// TwinCAT 3 PLC project PLC
// ProgramVersion: 3.1.4023.0
// libraries:
//   Tc2_Standard, * (Beckhoff Automation GmbH)
//   Tc2_System, * (Beckhoff Automation GmbH)
//   Tc3_Module, * (Beckhoff Automation GmbH)
// project tree:
//   / PlcTask.TcTTO
//   POUs/ MAIN.TcPOU
//   DUTs/IO/PdoEntries/ Status_57491DF1.TcDUT, Status_D4FDECD4.TcDUT, Control_0B2F8B70.TcDUT, Status_A3AA621F.TcDUT, Status_B0753356.TcDUT, Status_F2CE6D91.TcDUT, STATUS_B0753356.TcDUT, Status_8F1D55D8.TcDUT, Status_ACC8459F.TcDUT, Status_3A9E406C.TcDUT, Control_D500AB79.TcDUT, Status_D8D782C3.TcDUT, Control_6EF2C5D0.TcDUT, Status_E3E7FD12.TcDUT, Status_8CBE219F.TcDUT, Status_B6795845.TcDUT, Control_5FD4673D.TcDUT, Status_1E008DB9.TcDUT, Status_3035BE2E.TcDUT, Control_F189B737.TcDUT, Control_C948E0F2.TcDUT, Status_51F572C8.TcDUT
//   DUTs/IO/PDOs/ InfoData_6F19DB2B.TcDUT, Channel_830843C1.TcDUT, WcState_9091E0EB.TcDUT, ID_Inputs_07C9D28F.TcDUT, InfoData_32EB74EA.TcDUT, Latch_8E413295.TcDUT, WcState_B516A264.TcDUT, InfoData_A7436BC6.TcDUT, CNT_Input_Channel_FF10BD3C.TcDUT, DIG_Inputs_CAFF6004.TcDUT, DIG_Inputs_Device_1F4E72EB.TcDUT, CNT_Output_Channel_550BB6DF.TcDUT, DIG_Inputs_Channel_ACAA0425.TcDUT, DIG_Inputs_Channel_CC455148.TcDUT, DIG_Inputs_Channel_38F9DD27.TcDUT, AI_Inputs_Channel_C3DE7A0A.TcDUT, DIG_Inputs_Device_B3EA4204.TcDUT, Channel_42CA91F7.TcDUT, WcState_0B2B16F9.TcDUT, Diag_Channel_830843C1.TcDUT, DIG_Inputs_CC455148.TcDUT, DIG_Diag_Inputs_584303BF.TcDUT, DIG_Inputs_Device_E94E5BF9.TcDUT, DIG_Outputs_28AC1A9E.TcDUT, DIG_Outputs_Device_36A5EF17.TcDUT, DIG_Inputs_2D77DD63.TcDUT, DI_Inputs_Channel_91AC31B7.TcDUT, DO_Outputs_Channel_28AC1A9E.TcDUT, DIG_Diag_Inputs_Channel_584303BF.TcDUT, DIG_Output_Channel_28AC1A9E.TcDUT, DIG_Outputs_Channel_28AC1A9E.TcDUT, DIG_Inputs_Device_27CCC866.TcDUT, AI_Standard_Channel_A8DF64E3.TcDUT, RTD_RTDInputs_Channel_A8DF64E3.TcDUT, AI_Standard_Channel_4A394481.TcDUT, Ch1_Status_75824485.TcDUT, Ch1_Sample_A71DD501.TcDUT, Ch2_Status_75824485.TcDUT, Ch2_Sample_9F6886E6.TcDUT, NextSync1Time_9AFDC275.TcDUT, Sample_Count_EA88CAD9.TcDUT, InfoData_BEF6B88E.TcDUT, DIG_Inputs_697E0EF2.TcDUT, AI_Inputs_Channel_45213104.TcDUT, DEV_Inputs_Device_5F4E175E.TcDUT, DIG_Outputs_DE230DD5.TcDUT, DEV_Outputs_Device_59FFD247.TcDUT, AI_Inputs_Channel_5A86716D.TcDUT, AO_Output_Channel_BA7EBB7C.TcDUT, DI_Inputs_1F3A9325.TcDUT, AI_Inputs_Channel_A8DF64E3.TcDUT, SSI_Inputs_0E3D8E33.TcDUT, ENC_Status_compact_F4F89583.TcDUT, ENC_Control_compact_E6DC9B25.TcDUT, ENC_Status_compact_7D3464F3.TcDUT, ENC_Control_compact_21E2D14D.TcDUT, COM_Inputs_6C2FC202.TcDUT, COM_Outputs_5D00B5E7.TcDUT, COM_TxPDO_Map_Inputs_Channel_C252EAC2.TcDUT, COM_RxPDO_Map_Outputs_Channel_B336F4EE.TcDUT, COM_TxPDO_Map_Inputs_Channel_6C2FC202.TcDUT, COM_RxPDO_Map_Outputs_Channel_5D00B5E7.TcDUT, DIS_Inputs_E0E384E3.TcDUT, DIS_Outputs_6C9BFFEE.TcDUT, DeviceState_Inputs_Device_A1210598.TcDUT, DeviceState_Inputs_C7251DC9.TcDUT, Digital_Inputs_83D7E782.TcDUT, InfoData_90184F0C.TcDUT, Module_1_DeviceState_Inputs_Device_5322301C.TcDUT, Module_2_DeviceState_Inputs_B92A0D6A.TcDUT, Module_11_Digital_Inputs_33FD8372.TcDUT, ENC_Status_compact_4D066E1A.TcDUT, STM_Status_36ED096F.TcDUT, STM_Control_BA4CE352.TcDUT, STM_Velocity_A47A3F41.TcDUT, InfoData_6538CF5F.TcDUT, STM_Status_DE0D6B37.TcDUT, ENC_Status_compact_Channel_DC559AB0.TcDUT, DCM_Status_Channel_36ED096F.TcDUT, ENC_Control_compact_Channel_2E82BC43.TcDUT, DCM_Control_Channel_5A8B5016.TcDUT, DCM_Velocity_Channel_A47A3F41.TcDUT, InfoData_939F71B6.TcDUT, EPM_Inputs_Channel_B9246B8D.TcDUT, InfoData_E68C61CD.TcDUT, InfoData_2A97D6CF.TcDUT, Inputs_25A0042B.TcDUT, Outputs_2397A10E.TcDUT
//   DUTs/IO/Boxes/ EK1100_1FC0878B.TcDUT, EK1122_1FC0878B.TcDUT, EPP1004_D135F8DB.TcDUT, EPP1008_78E8D3DD.TcDUT, EPP1018_78E8D3DD.TcDUT, EPP1111_837A6B03.TcDUT, EPP1258_58F475DD.TcDUT, EPP1321_1FC0878B.TcDUT, EPP1322_1FC0878B.TcDUT, EPP1332_1FC0878B.TcDUT, EPP1342_1FC0878B.TcDUT, EPP1518_CC442588.TcDUT, EPP1809_32157CFD.TcDUT, EPP1819_32157CFD.TcDUT, EPP1816_73178B54.TcDUT, EPP1816_5E50D3DD.TcDUT, EPP1816_CABD51E6.TcDUT, EPP2008_E2806B95.TcDUT, EPP2028_E2806B95.TcDUT, EPP2038_3AE10DD7.TcDUT, EPP2304_47304899.TcDUT, EPP2308_F6D9A8D1.TcDUT, EPP2316_CAC4656D.TcDUT, EPP2316_D2866883.TcDUT, EPP2318_F6D9A8D1.TcDUT, EPP2328_F6D9A8D1.TcDUT, EPP2334_F6D9A8D1.TcDUT, EPP2338_7699BCF6.TcDUT, EPP2339_B2B612E8.TcDUT, EPP2339_8DFD1558.TcDUT, EPP2339_4CF33DED.TcDUT, EPP2349_8DFD1558.TcDUT, EPP2349_4CF33DED.TcDUT, EPP2624_7B64371E.TcDUT, EPP2809_2B6483BD.TcDUT, EPP2816_F9F6AB82.TcDUT, EPP2816_01296449.TcDUT, EPP2817_7CB3CE29.TcDUT, EPP3174_DCC78662.TcDUT, EPP3184_DCC78662.TcDUT, EPP3204_6CD7E119.TcDUT, EPP3204_AB25C3AC.TcDUT, EPP3314_E65CDB1C.TcDUT, EPP3632_E2B98A5C.TcDUT, EPP3744_315C92D4.TcDUT, EPP3752_C992DA1B.TcDUT, EPP4174_AB92710E.TcDUT, EPP4314_454AD8BA.TcDUT, EPP4374_A304750F.TcDUT, EPP5001_0B28D087.TcDUT, EPP5101_87AC78CF.TcDUT, EPP5101_7476E948.TcDUT, EPP5151_7476E948.TcDUT, EPP6001_40883D03.TcDUT, EPP6002_7F53816A.TcDUT, EPP6002_7BE6B617.TcDUT, EPP6090_18BD01E9.TcDUT, EPP6228_495B58F4.TcDUT, EPP7041_3210CF40.TcDUT, EPP7041_3E4BEAEF.TcDUT, EPP7342_2AE9C6B3.TcDUT, EPP9001_1FC0878B.TcDUT, EPP9022_32A9C19F.TcDUT
//   DUTs/IO/Devices/ SyncUnitTask_2D604ED5.TcDUT, SyncUnitTasks_6FEB8257.TcDUT, SyncUnits_99E584AF.TcDUT
//   DUTs/IO/Topology/ A_0024_EPP1342_0001_0017_FC9F5325.TcDUT, A_0023_EPP1342_0001_0016_822049EC.TcDUT, A_0022_EPP1332_0001_0017_EEFE2EB8.TcDUT, A_0021_EPP1332_0001_0016_54E1D1AE.TcDUT, A_0020_EPP1322_0001_0017_C93B3B41.TcDUT, A_0019_EPP1322_0001_0016_9024EDF1.TcDUT, A_0018_EPP1321_0060_0016_F908F4F3.TcDUT, Beckhoff_EPP1xxxEK1122_5ECABF39.TcDUT, Beckhoff_EPP1xxx_3250354D.TcDUT, Beckhoff_EPP2xxxEK1122_56176A05.TcDUT, Beckhoff_EPP2xxx_8ED37E64.TcDUT, Beckhoff_EPP3xxxEK1122_A76E71A7.TcDUT, Beckhoff_EPP3xxx_37FEE8A0.TcDUT, Beckhoff_EPP4xxxEK1122_FE2E0BEF.TcDUT, Beckhoff_EPP4xxx_F05B7AA2.TcDUT, Beckhoff_EPP5xxxEK1122_EF1F281E.TcDUT, Beckhoff_EPP5xxx_CECB1C9F.TcDUT, Beckhoff_EPP6xxxEK1122_484AACC3.TcDUT, Beckhoff_EPP6xxx_4A538F0B.TcDUT, Beckhoff_EPP7xxxEK1122_4AE68EFB.TcDUT, Beckhoff_EPP7xxx_26C654D6.TcDUT, Beckhoff_EPP9xxxEK1122_B72DCE23.TcDUT, Beckhoff_EPP9xxx_3F2579D7.TcDUT, EtherCAT_Master_EPPxxxx_9A8F5D7B.TcDUT
//   DUTs/IO/Base/ EtcSlaveBase_82538BE2.TcDUT, EtcSlaveBase_82538BE2.TcDUT, EtcSlaveBase_82538BE2.TcDUT, EtcSlaveTerminalBase_947E5A46.TcDUT, EtcSlaveBoxBase_77A0E4A7.TcDUT, EtcSlaveEndTerminalBase_866C7F0C.TcDUT, InputBase_8311D824.TcDUT, OutputBase_10CEE7DE.TcDUT, EtcMasterBase_62654B43.TcDUT
//   GVLs/ GVL_iXlinker.TcGVL
// real-time tasks:
//   TASK PlcTask: cycle T#10ms, priority 20, ADS port 350
// I/O:
//   DEVICE EtherCAT_Master_EPPxxxx, AmsNetId 172.20.30.238.13.1
//     Beckhoff EPP1xxx [EK1100 EtherCAT Coupler (2A E-Bus)]
//       Beckhoff EPP1xxxEK1122 [EK1122 2 port EtherCAT junction]
//         Beckhoff EPP1xxxsub EK1100 [EK1100 EtherCAT Coupler (2A E-Bus)]
//         A_0001(EPP1004-0061-0016) [EPP1004-0061 4 Ch. Dig. Input 24V, 3ms, M8]
//         A_0002(EPP1008-0001-0016) [EPP1008-0001 8 Ch. Dig. Input 24V, 3ms, M8]
//         A_0003(EPP1008-0001-0017) [EPP1008-0001 8 Ch. Dig. Input 24V, 3ms, M8]
//         A_0004(EPP1008-0002-0016) [EPP1008-0002 8 Ch. Dig. Input 24V, 3ms, M12]
//         A_0005(EPP1008-0002-0017) [EPP1008-0002 8 Ch. Dig. Input 24V, 3ms, M12]
//         A_0006(EPP1008-0022-0016) [EPP1008-0022 8 Ch. Dig. Input 24V, 3ms, M12]
//         A_0007(EPP1018-0001-0016) [EPP1018-0001 8 Ch. Dig. Input 24V, 10µs, M8]
//         A_0008(EPP1018-0001-0017) [EPP1018-0001 8 Ch. Dig. Input 24V, 10µs, M8]
//         A_0009(EPP1018-0002-0016) [EPP1018-0002 8 Ch. Dig. Input 24V, 10µs, M12]
//         A_0010(EPP1018-0002-0017) [EPP1018-0002 8 Ch. Dig. Input 24V, 10µs, M12]
//         A_0011(EPP1111-0000-0016) [EPP1111-0000 ID-Switch]
//         A_0012(EPP1111-0000-0017) [EPP1111-0000 ID-Switch]
//         A_0013(EPP1111-0000-0018) [EPP1111-0000 ID-Switch]
//         A_0014(EPP1258-0001-0016) [EPP1258-0001 8 Ch. Dig. Input 24V, 10µs, DC Latch, M8]
//         A_0015(EPP1258-0001-0017) [EPP1258-0001 8 Ch. Dig. Input 24V, 10µs, DC Latch, M8]
//         A_0016(EPP1258-0002-0016) [EPP1258-0002 8 Ch. Dig. Input 24V, 10µs, DC Latch, M12]
//         A_0017(EPP1258-0002-0017) [EPP1258-0002 8 Ch. Dig. Input 24V, 10µs, DC Latch, M12]
//         A_0018(EPP1321-0060-0016) [EPP1321-0060 1 port EtherCAT P gateway]
//           A_0019(EPP1322-0001-0016) [EPP1322-0001 3 port EtherCAT P gateway]
//             A_0020(EPP1322-0001-0017) [EPP1322-0001 3 port EtherCAT P gateway]
//               A_0021(EPP1332-0001-0016) [EPP1332-0001 3 port EtherCAT P junction, power refreshing]
//                 A_0022(EPP1332-0001-0017) [EPP1332-0001 3 port EtherCAT P junction, power refreshing]
//                   A_0023(EPP1342-0001-0016) [EPP1342-0001 3 port EtherCAT P junction]
//                     A_0024(EPP1342-0001-0017) [EPP1342-0001 3 port EtherCAT P junction]
//                       A_0025(EPP1518-0002-0016) [EPP1518-0002 8 Ch.digital multi-function input]
//                       A_0026(EPP1518-0002-0017) [EPP1518-0002 8 Ch.digital multi-function input]
//                       A_0027(EPP1809-0021-0016) [EPP1809-0021 16 Ch. Dig. Input 24V, 3ms, M8]
//                       A_0028(EPP1809-0022-0016) [EPP1809-0022 16 Ch. Dig. Input 24V, 3ms, M8]
//                       A_0029(EPP1819-0021-0016) [EPP1819-0021 16 Ch. Dig. Input 24V, 10µs, M8]
//                       A_0030(EPP1819-0022-0016) [EPP1819-0022 16 Ch. Dig. Input 24V, 10µs, M8]
//                       A_0031(EPP1816-0003-0016) [EPP1816-0003 16 Ch. Dig. Input 24V, 10µs, 10-Pole Plug Connector]
//                       A_0032(EPP1816-0008-0016) [EPP1816-0008 16 Ch. Dig. Input 24V, 10µs, D-SUB25]
//                       A_0033(EPP1816-0008-0017) [EPP1816-0008 16 Ch. Dig. Input 24V, 10µs, D-SUB25]
//                       A_0034(EPP1816-0008-0018) [EPP1816-0008 16 Ch. Dig. Input 24V, 10µs, D-SUB25]
//                       A_0035(EPP1816-3008-0016) [EPP1816-3008 16Ch. Dig. Input  24V 10µs Acceleration Sensor, DSUB-25]
//     Beckhoff EPP2xxx [EK1100 EtherCAT Coupler (2A E-Bus)]
//       Beckhoff EPP2xxxEK1122 [EK1122 2 port EtherCAT junction]
//         Beckhoff EPP2xxxsub EK1100 [EK1100 EtherCAT Coupler (2A E-Bus)]
//         A_0001(EPP2008-0001-0016) [EPP2008-0001 8 Ch. Dig. Output 24V, 0,5A, M8]
//         A_0002(EPP2008-0001-0017) [EPP2008-0001 8 Ch. Dig. Output 24V, 0,5A, M8]
//         A_0003(EPP2008-0001-0018) [EPP2008-0001 8 Ch. Dig. Output 24V, 0,5A, M8]
//         A_0004(EPP2008-0002-0016) [EPP2008-0002 8 Ch. Dig. Output 24V, 0,5A, M12]
//         A_0005(EPP2008-0002-0017) [EPP2008-0002 8 Ch. Dig. Output 24V, 0,5A, M12]
//         A_0006(EPP2008-0002-0018) [EPP2008-0002 8 Ch. Dig. Output 24V, 0,5A, M12]
//         A_0007(EPP2008-0022-0016) [EPP2008-0022 8 Ch. Dig. Output 24V, 0,5A, M12]
//         A_0008(EPP2028-0001-0016) [EPP2028-0001 8 Ch. Dig. Output 24V, 2A, M8]
//         A_0009(EPP2028-0001-0017) [EPP2028-0001 8 Ch. Dig. Output 24V, 2A, M8]
//         A_0010(EPP2028-0002-0016) [EPP2028-0002 8 Ch. Dig. Output 24V, 2A, M12]
//         A_0011(EPP2028-0002-0017) [EPP2028-0002 8 Ch. Dig. Output 24V, 2A, M12]
//         A_0012(EPP2038-0001-0016) [EPP2038-0001 8 Ch. Dig. Output 24V, 2A, M8, Diagnostic]
//         A_0013(EPP2038-0002-0016) [EPP2038-0002 8 Ch. Dig. Output 24V, 2A, M8, Diagnostic]
//         A_0014(EPP2304-0061-0016) [EPP2304-0061 2 CH. Dig. In, 3ms, 2 Ch. Dig. Out 24V, 0,5A, M12]
//         A_0015(EPP2304-0061-0017) [EPP2304-0061 2 CH. Dig. In, 3ms, 2 Ch. Dig. Out 24V, 0,5A, M12]
//         A_0016(EPP2304-0061-0018) [EPP2304-0061 2 CH. Dig. In, 3ms, 2 Ch. Dig. Out 24V, 0,5A, M12]
//         A_0017(EPP2308-0001-0016) [EPP2308-0001 4 Ch. Dig. In, 3ms, 4 Ch. Dig. Out 24V, 0,5A, M8]
//         A_0018(EPP2308-0001-0017) [EPP2308-0001 4 Ch. Dig. In, 3ms, 4 Ch. Dig. Out 24V, 0,5A, M8]
//         A_0019(EPP2308-0001-0018) [EPP2308-0001 4 Ch. Dig. In, 3ms, 4 Ch. Dig. Out 24V, 0,5A, M8]
//         A_0020(EPP2308-0002-0016) [EPP2308-0002 4 CH. Dig. In, 3ms, 4 Ch. Dig. Out 24V, 0,5A, M12]
//         A_0021(EPP2308-0002-0017) [EPP2308-0002 4 CH. Dig. In, 3ms, 4 Ch. Dig. Out 24V, 0,5A, M12]
//         A_0022(EPP2308-0002-0018) [EPP2308-0002 4 CH. Dig. In, 3ms, 4 Ch. Dig. Out 24V, 0,5A, M12]
//         A_0023(EPP2316-0003-0016) [EPP2316-0003 8 Ch. Dig. In, 10µs, 8Ch. Dig. Out 24V, 0,5A, Diagnostic, 10-Pole Plug Connector]
//         A_0024(EPP2316-0003-0017) [EPP2316-0003 8 Ch. Dig. In, 10µs, 8Ch. Dig. Out 24V, 0,5A, Diagnostic, 10-Pole Plug Connector]
//         A_0025(EPP2316-0003-0018) [EPP2316-0003 8 Ch. Dig. In, 10µs, 8Ch. Dig. Out 24V, 0,5A, Diagnostic, 10-Pole Plug Connector]
//         A_0026(EPP2316-0008-0016) [EPP2316-0008 8 Ch. Dig. In, 10µs, 8Ch. Dig. Out 24V, 0,5A, Diagnostic, D-SUB25]
//         A_0027(EPP2316-0008-0017) [EPP2316-0008 8 Ch. Dig. In, 10µs, 8Ch. Dig. Out 24V, 0,5A, Diagnostic, D-SUB25]
//         A_0028(EPP2316-0008-0018) [EPP2316-0008 8 Ch. Dig. In, 10µs, 8Ch. Dig. Out 24V, 0,5A, Diagnostic, D-SUB25]
//         A_0029(EPP2318-0001-0016) [EPP2318-0001 4 Ch. Dig. In, 10µs, 4 Ch. Dig. Out 24V, 0,5A, M8]
//         A_0030(EPP2318-0001-0017) [EPP2318-0001 4 Ch. Dig. In, 10µs, 4 Ch. Dig. Out 24V, 0,5A, M8]
//         A_0031(EPP2318-0001-0018) [EPP2318-0001 4 Ch. Dig. In, 10µs, 4 Ch. Dig. Out 24V, 0,5A, M8]
//         A_0032(EPP2318-0002-0016) [EPP2318-0002 4 Ch. Dig. In, 10µs, 4 Ch. Dig. Out 24V, 0,5A, M12]
//         A_0033(EPP2318-0002-0017) [EPP2318-0002 4 Ch. Dig. In, 10µs, 4 Ch. Dig. Out 24V, 0,5A, M12]
//         A_0034(EPP2318-0002-0018) [EPP2318-0002 4 Ch. Dig. In, 10µs, 4 Ch. Dig. Out 24V, 0,5A, M12]
//         A_0035(EPP2328-0001-0016) [EPP2328-0001 4 CH. Dig. In, 3ms, 4 Ch. Dig. Out 24V, 2A, M8]
//         A_0036(EPP2328-0001-0017) [EPP2328-0001 4 CH. Dig. In, 3ms, 4 Ch. Dig. Out 24V, 2A, M8]
//         A_0037(EPP2328-0001-0018) [EPP2328-0001 4 CH. Dig. In, 3ms, 4 Ch. Dig. Out 24V, 2A, M8]
//         A_0038(EPP2328-0002-0016) [EPP2328-0002 4 CH. Dig. In, 3ms, 4 Ch. Dig. Out 24V, 2A, M12]
//         A_0039(EPP2328-0002-0017) [EPP2328-0002 4 CH. Dig. In, 3ms, 4 Ch. Dig. Out 24V, 2A, M12]
//         A_0040(EPP2328-0002-0018) [EPP2328-0002 4 CH. Dig. In, 3ms, 4 Ch. Dig. Out 24V, 2A, M12]
//         A_0041(EPP2334-0061-0016) [EPP2334-0061 4 Ch. Dig. Input/Output 24V, 0,5A, M8]
//         A_0042(EPP2334-0061-0017) [EPP2334-0061 4 Ch. Dig. Input/Output 24V, 0,5A, M8]
//         A_0043(EPP2334-0061-0018) [EPP2334-0061 4 Ch. Dig. Input/Output 24V, 0,5A, M8]
//         A_0044(EPP2334-0061-0019) [EPP2334-0061 4 Ch. Dig. Input/Output 24V, 0,5A, M8]
//         A_0045(EPP2338-0001-0016) [EPP2338-0001 8 Ch. Dig. Input/Output 24V, 0,5A, M8]
//         A_0046(EPP2338-0001-0017) [EPP2338-0001 8 Ch. Dig. Input/Output 24V, 0,5A, M8]
//         A_0047(EPP2338-0001-0018) [EPP2338-0001 8 Ch. Dig. Input/Output 24V, 0,5A, M8]
//         A_0048(EPP2338-0002-0016) [EPP2338-0002 8 Ch. Dig. Input/Output 24V, 0,5A, M12]
//         A_0049(EPP2338-0002-0017) [EPP2338-0002 8 Ch. Dig. Input/Output 24V, 0,5A, M12]
//         A_0050(EPP2338-0002-0018) [EPP2338-0002 8 Ch. Dig. Input/Output 24V, 0,5A, M12]
//         A_0051(EPP2338-1001-0017) [EPP2338-1001 8 Ch. Dig. Input/Output 24V, 3ms, 0,5A, M8]
//         A_0052(EPP2338-1001-0018) [EPP2338-1001 8 Ch. Dig. Input/Output 24V, 3ms, 0,5A, M8]
//         A_0053(EPP2338-1001-0019) [EPP2338-1001 8 Ch. Dig. Input/Output 24V, 3ms, 0,5A, M8]
//         A_0054(EPP2338-1002-0017) [EPP2338-1002 8 Ch. Dig. Input/Output 24V, 3ms, 0,5A, M12]
//         A_0055(EPP2338-1002-0018) [EPP2338-1002 8 Ch. Dig. Input/Output 24V, 3ms, 0,5A, M12]
//         A_0056(EPP2338-1002-0019) [EPP2338-1002 8 Ch. Dig. Input/Output 24V, 3ms, 0,5A, M12]
//         A_0057(EPP2339-0003-0016) [EPP2339-0003 16 Ch. Dig. Input/Output 24V, 0,5A, 10-Pole Plug Connector]
//         A_0058(EPP2339-0021-0016) [EPP2339-0021 16 Ch. Dig. Input/Output 24V, 0,5A, M8]
//         A_0059(EPP2339-0021-0017) [EPP2339-0021 16 Ch. Dig. Input/Output 24V, 0,5A, M8]
//         A_0060(EPP2339-0021-0018) [EPP2339-0021 16 Ch. Dig. Input/Output 24V, 0,5A, M8]
//         A_0061(EPP2339-0022-0016) [EPP2339-0022 16 Ch. Dig. Input/Output 24V, 0,5A, M8]
//         A_0062(EPP2339-0022-0017) [EPP2339-0022 16 Ch. Dig. Input/Output 24V, 0,5A, M8]
//         A_0063(EPP2339-0022-0018) [EPP2339-0022 16 Ch. Dig. Input/Output 24V, 0,5A, M8]
//         A_0064(EPP2349-0021-0016) [EPP2349-0021 16 Ch. Dig. Input/Output 24V, 10µs, 0,5A, M8]
//         A_0065(EPP2349-0021-0017) [EPP2349-0021 16 Ch. Dig. Input/Output 24V, 10µs, 0,5A, M8]
//         A_0066(EPP2349-0021-0018) [EPP2349-0021 16 Ch. Dig. Input/Output 24V, 10µs, 0,5A, M8]
//         A_0067(EPP2349-0022-0016) [EPP2349-0022 16 Ch. Dig. Input/Output 24V, 10µs, 0,5A, M8]
//         A_0068(EPP2349-0022-0017) [EPP2349-0022 16 Ch. Dig. Input/Output 24V, 10µs, 0,5A, M8]
//         A_0069(EPP2349-0022-0018) [EPP2349-0022 16 Ch. Dig. Input/Output 24V, 10µs, 0,5A, M8]
//         A_0070(EPP2624-0002-0016) [EPP2624-0002 4Ch. Relay Output, NO (125V AC / 30V DC)]
//         A_0071(EPP2809-0021-0016) [EPP2809-0021 16 Ch. Dig. Output 24V, 0,5A, M8]
//         A_0072(EPP2809-0022-0016) [EPP2809-0022 16 Ch. Dig. Output 24V, 0,5A, M8]
//         A_0073(EPP2816-0004-0016) [EPP2816-0004 16CH. Dig. Output, Diagnostic, M16]
//         A_0074(EPP2816-0004-0017) [EPP2816-0004 16CH. Dig. Output, Diagnostic, M16]
//         A_0075(EPP2816-0008-0016) [EPP2816-0008 16 Ch. Dig. Output 24V, 0,5A, Diagnostic, D-SUB25]
//         A_0076(EPP2816-0008-0017) [EPP2816-0008 16 Ch. Dig. Output 24V, 0,5A, Diagnostic, D-SUB25]
//         A_0077(EPP2816-0008-0018) [EPP2816-0008 16 Ch. Dig. Output 24V, 0,5A, Diagnostic, D-SUB25]
//         A_0078(EPP2816-0010-0016) [EPP2816-0010 16 Ch. Dig. Output 24V, 0,5A, Diagnostic, D-SUB9]
//         A_0079(EPP2816-0010-0017) [EPP2816-0010 16 Ch. Dig. Output 24V, 0,5A, Diagnostic, D-SUB9]
//         A_0080(EPP2816-0010-0018) [EPP2816-0010 16 Ch. Dig. Output 24V, 0,5A, Diagnostic, D-SUB9]
//         A_0081(EPP2817-0008-0016) [EPP2817-0008 24Ch. Dig. Output 24V 0,5A, Diagnostics, DSUB-25]
//         A_0082(EPP2817-0008-0017) [EPP2817-0008 24Ch. Dig. Output 24V 0,5A, Diagnostics, DSUB-25]
//         A_0083(EPP2817-0008-0018) [EPP2817-0008 24Ch. Dig. Output 24V 0,5A, Diagnostics, DSUB-25]
//     Beckhoff EPP3xxx [EK1100 EtherCAT Coupler (2A E-Bus)]
//       Beckhoff EPP3xxxEK1122 [EK1122 2 port EtherCAT junction]
//         Beckhoff EPP3xxxsub EK1100 [EK1100 EtherCAT Coupler (2A E-Bus)]
//         A_0001(EPP3174-0002-0016) [EPP3174-0002 4Ch. Ana. Input +/-10V, 0-10V, 0/4-20mA configurable]
//         A_0002(EPP3174-0002-0017) [EPP3174-0002 4Ch. Ana. Input +/-10V, 0-10V, 0/4-20mA configurable]
//         A_0003(EPP3174-0002-0018) [EPP3174-0002 4Ch. Ana. Input +/-10V, 0-10V, 0/4-20mA configurable]
//         A_0004(EPP3184-0002-0016) [EPP3184-0002 4Ch. Ana. Input +/-10V, 0-10V, 0/4-20mA configurable, single ended]
//         A_0005(EPP3184-0002-0017) [EPP3184-0002 4Ch. Ana. Input +/-10V, 0-10V, 0/4-20mA configurable, single ended]
//         A_0006(EPP3184-0002-0018) [EPP3184-0002 4Ch. Ana. Input +/-10V, 0-10V, 0/4-20mA configurable, single ended]
//         A_0007(EPP3184-0002-0019) [EPP3184-0002 4Ch. Ana. Input +/-10V, 0-10V, 0/4-20mA configurable, single ended]
//         A_0008(EPP3204-0002-0016) [EPP3204-0002 4Ch. Ana. Input PT100 (RTD)]
//         A_0009(EPP3204-0002-0017) [EPP3204-0002 4Ch. Ana. Input PT100 (RTD)]
//         A_0010(EPP3204-0002-0018) [EPP3204-0002 4Ch. Ana. Input PT100 (RTD)]
//         A_0011(EPP3204-0002-0019) [EPP3204-0002 4Ch. Ana. Input PT100 (RTD)]
//         A_0012(EPP3314-0002-0016) [EPP3314-0002 4Ch. Ana. Input Thermocouple (TC)]
//         A_0013(EPP3314-0002-0017) [EPP3314-0002 4Ch. Ana. Input Thermocouple (TC)]
//         A_0014(EPP3314-0002-0018) [EPP3314-0002 4Ch. Ana. Input Thermocouple (TC)]
//         A_0015(EPP3632-0001-0016) [EPP3632-0001 2Ch. IEPE Sensor]
//         A_0016(EPP3632-0001-0017) [EPP3632-0001 2Ch. IEPE Sensor]
//         A_0017(EPP3744-0041-0016) [EPP3744-0041 5Ch. Absolute Pressure 6Ch. Dig. Input 10us 2Ch. Dig. Output 24V 0,5A M8]
//         A_0018(EPP3744-0041-0017) [EPP3744-0041 5Ch. Absolute Pressure 6Ch. Dig. Input 10us 2Ch. Dig. Output 24V 0,5A M8]
//         A_0019(EPP3744-0041-0018) [EPP3744-0041 5Ch. Absolute Pressure 1Bar 6Ch. Dig. Input 10us 2Ch. Dig. Output 24V 0,5A M8]
//         A_0020(EPP3744-1041-0016) [EPP3744-1041 5Ch. Absolute Pressure 6Ch. Dig. Input 10us 2Ch. Dig. Output 24V 0,5A M8]
//         A_0021(EPP3744-1041-0017) [EPP3744-1041 5Ch. Absolute Pressure 6Ch. Dig. Input 10us 2Ch. Dig. Output 24V 0,5A M8]
//         A_0022(EPP3744-1041-0018) [EPP3744-1041 5Ch. Absolute Pressure 6Ch. Dig. Input 10us 2Ch. Dig. Output 24V 0,5A M8]
//         A_0023(EPP3744-1041-0019) [EPP3744-1041 5Ch. Absolute Pressure 7Bar 6Ch. Dig. Input 10us 2Ch. Dig. Output 24V 0,5A M8]
//         A_0024(EPP3744-1041-0020) [EPP3744-1041 5Ch. Absolute Pressure 7Bar 6Ch. Dig. Input 10us 2Ch. Dig. Output 24V 0,5A M8]
//         A_0025(EPP3752-0000-0017) [EPP3752-0000 Acceleration Sensor]
//     Beckhoff EPP4xxx [EK1100 EtherCAT Coupler (2A E-Bus)]
//       Beckhoff EPP4xxxEK1122 [EK1122 2 port EtherCAT junction]
//         Beckhoff EPP4xxxsub EK1100 [EK1100 EtherCAT Coupler (2A E-Bus)]
//         A_0001(EPP4174-0002-0016) [EPP4174-0002 4Ch. Ana. Output +/-10V, 0-10V, 0/4-20mA configurable]
//         A_0002(EPP4174-0002-0017) [EPP4174-0002 4Ch. Ana. Output +/-10V, 0-10V, 0/4-20mA configurable]
//         A_0003(EPP4314-1002-0016) [EPP4314-1002 2Ch. Ana. Input -20/0/4-20mA; 2Ch. Ana. Output -20/0/4-20mA configurable]
//         A_0004(EPP4374-0002-0016) [EPP4374-0002 2Ch. Ana. Input +/-10V, 0-10V, 0/4-20mA configurable; 2Ch. Ana. Output +/-10V, 0-10V, 0/4-20mA configurable]
//         A_0005(EPP4374-0002-0017) [EPP4374-0002 2Ch. Ana. Input +/-10V, 0-10V, 0/4-20mA configurable; 2Ch. Ana. Output +/-10V, 0-10V, 0/4-20mA configurable]
//         A_0006(EPP4374-0002-0018) [EPP4374-0002 2Ch. Ana. Input +/-10V, 0-10V, 0/4-20mA configurable; 2Ch. Ana. Output +/-10V, 0-10V, 0/4-20mA configurable]
//         A_0007(EPP4374-0002-0019) [EPP4374-0002 2Ch. Ana. Input +/-10V, 0-10V, 0/4-20mA configurable; 2Ch. Ana. Output +/-10V, 0-10V, 0/4-20mA configurable]
//     Beckhoff EPP5xxx [EK1100 EtherCAT Coupler (2A E-Bus)]
//       Beckhoff EPP5xxxEK1122 [EK1122 2 port EtherCAT junction]
//         Beckhoff EPP5xxxsub EK1100 [EK1100 EtherCAT Coupler (2A E-Bus)]
//         A_0001(EPP5001-0002-0016) [EPP5001-0002 1Ch. SSI Encoder]
//         A_0002(EPP5101-0002-0016) [EPP5101-0002 1Ch. Inc. Encoder 5V, M12]
//         A_0003(EPP5101-0002-0017) [EPP5101-0002 1Ch. Inc. Encoder 5V, M12]
//         A_0004(EPP5101-0011-0016) [EPP5101-0011 1Ch. Inc. Encoder 5V, D-SUB15]
//         A_0005(EPP5101-0011-0017) [EPP5101-0011 1Ch. Inc. Encoder 5V, D-SUB15]
//         A_0006(EPP5101-1002-0016) [EPP5101-1002 1Ch. Inc. Encoder 5V, M12, 24V Sensor Supply]
//         A_0007(EPP5101-1002-0017) [EPP5101-1002 1Ch. Inc. Encoder 5V, M12, 24V Sensor Supply]
//         A_0008(EPP5151-0002-0016) [EPP5151-0002 1Ch. Inc. Encoder 24V, M12, single ended]
//         A_0009(EPP5151-0002-0017) [EPP5151-0002 1Ch. Inc. Encoder 24V, M12, single ended]
//     Beckhoff EPP6xxx [EK1100 EtherCAT Coupler (2A E-Bus)]
//       Beckhoff EPP6xxxEK1122 [EK1122 2 port EtherCAT junction]
//         Beckhoff EPP6xxxsub EK1100 [EK1100 EtherCAT Coupler (2A E-Bus)]
//         A_0001(EPP6001-0002-0016) [EPP6001-0002 Interface (RS232/422/485)]
//         A_0002(EPP6001-0002-0017) [EPP6001-0002 Interface (RS232/422/485)]
//         A_0003(EPP6001-0002-0018) [EPP6001-0002 Interface (RS232/422/485)]
//         A_0004(EPP6002-0002-0016) [EPP6002-0002 Interface (RS232/422/485)]
//         A_0005(EPP6002-0002-0017) [EPP6002-0002 Interface (RS232/422/485)]
//         A_0006(EPP6002-0002-0018) [EPP6002-0002 Interface (RS232/422/485)]
//         A_0007(EPP6002-0002-0019) [EPP6002-0002 Interface (RS232/422/485)]
//         A_0008(EPP6090-0000-0017) [EPP6090 Display box]
//         A_0009(EPP6228-0022-0016) [EPP6228 (IO Link Master)]
//           modules: Module 1 (DeviceState Inputs Device), Module 2 (DeviceState Inputs), Module 3 (empty), Module 4 (empty), Module 5 (empty), Module 6 (empty), Module 7 (empty), Module 8 (empty), Module 9 (empty), Module 10 (empty), Module 11 (Digital Inputs)
//     Beckhoff EPP7xxx [EK1100 EtherCAT Coupler (2A E-Bus)]
//       Beckhoff EPP7xxxEK1122 [EK1122 2 port EtherCAT junction]
//         Beckhoff EPP7xxxsub EK1100 [EK1100 EtherCAT Coupler (2A E-Bus)]
//         A_0001(EPP7041-1002-0016) [EPP7041-1002 1Ch. Stepper motor output stage (50V, 1.5A)]
//         A_0002(EPP7041-1002-0017) [EPP7041-1002 1Ch. Stepper motor output stage (50V, 1.5A)]
//         A_0003(EPP7041-1002-0023) [EPP7041-1002 1Ch. Stepper motor output stage (50V, 1.5A)]
//         A_0004(EPP7041-3002-0016) [EPP7041-3002 1Ch. Stepper motor output stage (50V, 5A)]
//         A_0005(EPP7041-3002-0017) [EPP7041-3002 1Ch. Stepper motor output stage (50V, 5A)]
//         A_0006(EPP7041-3002-0018) [EPP7041-3002 1Ch. Stepper motor output stage (50V, 5A)]
//         A_0007(EPP7041-3002-0023) [EPP7041-3002 1Ch. Stepper motor output stage (50V, 5A)]
//         A_0008(EPP7342-0002-0016) [EPP7342-0002 2Ch. DC motor output stage (50V, 3.5A)]
//         A_0009(EPP7342-0002-0017) [EPP7342-0002 2Ch. DC motor output stage (50V, 3.5A)]
//     Beckhoff EPP9xxx [EK1100 EtherCAT Coupler (2A E-Bus)]
//       Beckhoff EPP9xxxEK1122 [EK1122 2 port EtherCAT junction]
//         Beckhoff EPP9xxxsub EK1100 [EK1100 EtherCAT Coupler (2A E-Bus)]
//         A_0001(EPP9001-0060-0016) [EPP9001-0060 4 K. Dig. EtherCAT P / EtherCAT ECP/EC Connector with voltage forwarding]
//         A_0002(EPP9001-0060-0017) [EPP9001-0060 4 K. Dig. EtherCAT P / EtherCAT ECP/EC Connector with voltage forwarding]
//         A_0003(EPP9022-0060-0017) [EPP9022-0060 ECat P Diagnostic Box]
//         A_0004(EPP9022-9060-0017) [EPP9022-9060 ECat P Diagnostic Box, TwinSAFE SC]
// variable links:
//   PLC/PLC Instance <-> EtherCAT Master EPPxxxx/Beckhoff EPP1xxx
//     PlcTask Inputs/GVL_iXlinker.EtherCAT_Master_EPPxxxx.Beckhoff_EPP1xxx.InfoData.State <-> InfoData/State
//   PLC/PLC Instance <-> EtherCAT Master EPPxxxx/Beckhoff EPP1xxx/Beckhoff EPP1xxxEK1122
//     PlcTask Inputs/GVL_iXlinker.EtherCAT_Master_EPPxxxx.Beckhoff_EPP1xxx.Beckhoff_EPP1xxxEK1122.InfoData.State <-> InfoData/State
//   PLC/PLC Instance <-> EtherCAT Master EPPxxxx/Beckhoff EPP1xxx/Beckhoff EPP1xxxEK1122/Beckhoff EPP1xxxsub EK1100
//     PlcTask Inputs/GVL_iXlinker.EtherCAT_Master_EPPxxxx.Beckhoff_EPP1xxx.Beckhoff_EPP1xxxEK1122.Beckhoff_EPP1xxxsub_EK1100.InfoData.State <-> InfoData/State
//   PLC/PLC Instance <-> EtherCAT Master EPPxxxx/Beckhoff EPP1xxx/Beckhoff EPP1xxxEK1122/A_0001(EPP1004-0061-0016)
//     PlcTask Inputs/GVL_iXlinker.EtherCAT_Master_EPPxxxx.Beckhoff_EPP1xxx.Beckhoff_EPP1xxxEK1122.A_0001_EPP1004_0061_0016.Channel_1.Input <-> Channel 1/Input
//     PlcTask Inputs/GVL_iXlinker.EtherCAT_Master_EPPxxxx.Beckhoff_EPP1xxx.Beckhoff_EPP1xxxEK1122.A_0001_EPP1004_0061_0016.Channel_2.Input <-> Channel 2/Input
//     PlcTask Inputs/GVL_iXlinker.EtherCAT_Master_EPPxxxx.Beckhoff_EPP1xxx.Beckhoff_EPP1xxxEK1122.A_0001_EPP1004_0061_0016.Channel_3.Input <-> Channel 3/Input
//     PlcTask Inputs/GVL_iXlinker.EtherCAT_Master_EPPxxxx.Beckhoff_EPP1xxx.Beckhoff_EPP1xxxEK1122.A_0001_EPP1004_0061_0016.Channel_4.Input <-> Channel 4/Input
//     PlcTask Inputs/GVL_iXlinker.EtherCAT_Master_EPPxxxx.Beckhoff_EPP1xxx.Beckhoff_EPP1xxxEK1122.A_0001_EPP1004_0061_0016.WcState.WcState <-> WcState/WcState
//     PlcTask Inputs/GVL_iXlinker.EtherCAT_Master_EPPxxxx.Beckhoff_EPP1xxx.Beckhoff_EPP1xxxEK1122.A_0001_EPP1004_0061_0016.WcState.InputToggle <-> WcState/InputToggle
//     PlcTask Inputs/GVL_iXlinker.EtherCAT_Master_EPPxxxx.Beckhoff_EPP1xxx.Beckhoff_EPP1xxxEK1122.A_0001_EPP1004_0061_0016.InfoData.State <-> InfoData/State
//   PLC/PLC Instance <-> EtherCAT Master EPPxxxx/Beckhoff EPP1xxx/Beckhoff EPP1xxxEK1122/A_0002(EPP1008-0001-0016)
//     PlcTask Inputs/GVL_iXlinker.EtherCAT_Master_EPPxxxx.Beckhoff_EPP1xxx.Beckhoff_EPP1xxxEK1122.A_0002_EPP1008_0001_0016.Channel_1.Input <-> Channel 1/Input
//     PlcTask Inputs/GVL_iXlinker.EtherCAT_Master_EPPxxxx.Beckhoff_EPP1xxx.Beckhoff_EPP1xxxEK1122.A_0002_EPP1008_0001_0016.Channel_2.Input <-> Channel 2/Input
//     PlcTask Inputs/GVL_iXlinker.EtherCAT_Master_EPPxxxx.Beckhoff_EPP1xxx.Beckhoff_EPP1xxxEK1122.A_0002_EPP1008_0001_0016.Channel_3.Input <-> Channel 3/Input
//     PlcTask Inputs/GVL_iXlinker.EtherCAT_Master_EPPxxxx.Beckhoff_EPP1xxx.Beckhoff_EPP1xxxEK1122.A_0002_EPP1008_0001_0016.Channel_4.Input <-> Channel 4/Input
//     PlcTask Inputs/GVL_iXlinker.EtherCAT_Master_EPPxxxx.Beckhoff_EPP1xxx.Beckhoff_EPP1xxxEK1122.A_0002_EPP1008_0001_0016.Channel_5.Input <-> Channel 5/Input
//     PlcTask Inputs/GVL_iXlinker.EtherCAT_Master_EPPxxxx.Beckhoff_EPP1xxx.Beckhoff_EPP1xxxEK1122.A_0002_EPP1008_0001_0016.Channel_6.Input <-> Channel 6/Input
//     PlcTask Inputs/GVL_iXlinker.EtherCAT_Master_EPPxxxx.Beckhoff_EPP1xxx.Beckhoff_EPP1xxxEK1122.A_0002_EPP1008_0001_0016.Channel_7.Input <-> Channel 7/Input
//     PlcTask Inputs/GVL_iXlinker.EtherCAT_Master_EPPxxxx.Beckhoff_EPP1xxx.Beckhoff_EPP1xxxEK1122.A_0002_EPP1008_0001_0016.Channel_8.Input <-> Channel 8/Input
//     PlcTask Inputs/GVL_iXlinker.EtherCAT_Master_EPPxxxx.Beckhoff_EPP1xxx.Beckhoff_EPP1xxxEK1122.A_0002_EPP1008_0001_0016.WcState.WcState <-> WcState/WcState
//     PlcTask Inputs/GVL_iXlinker.EtherCAT_Master_EPPxxxx.Beckhoff_EPP1xxx.Beckhoff_EPP1xxxEK1122.A_0002_EPP1008_0001_0016.WcState.InputToggle <-> WcState/InputToggle
//     PlcTask Inputs/GVL_iXlinker.EtherCAT_Master_EPPxxxx.Beckhoff_EPP1xxx.Beckhoff_EPP1xxxEK1122.A_0002_EPP1008_0001_0016.InfoData.State <-> InfoData/State
//   PLC/PLC Instance <-> EtherCAT Master EPPxxxx/Beckhoff EPP1xxx/Beckhoff EPP1xxxEK1122/A_0003(EPP1008-0001-0017)
//     PlcTask Inputs/GVL_iXlinker.EtherCAT_Master_EPPxxxx.Beckhoff_EPP1xxx.Beckhoff_EPP1xxxEK1122.A_0003_EPP1008_0001_0017.Channel_1.Input <-> Channel 1/Input
//     PlcTask Inputs/GVL_iXlinker.EtherCAT_Master_EPPxxxx.Beckhoff_EPP1xxx.Beckhoff_EPP1xxxEK1122.A_0003_EPP1008_0001_0017.Channel_2.Input <-> Channel 2/Input
//     PlcTask Inputs/GVL_iXlinker.EtherCAT_Master_EPPxxxx.Beckhoff_EPP1xxx.Beckhoff_EPP1xxxEK1122.A_0003_EPP1008_0001_0017.Channel_3.Input <-> Channel 3/Input
//     PlcTask Inputs/GVL_iXlinker.EtherCAT_Master_EPPxxxx.Beckhoff_EPP1xxx.Beckhoff_EPP1xxxEK1122.A_0003_EPP1008_0001_0017.Channel_4.Input <-> Channel 4/Input
//     PlcTask Inputs/GVL_iXlinker.EtherCAT_Master_EPPxxxx.Beckhoff_EPP1xxx.Beckhoff_EPP1xxxEK1122.A_0003_EPP1008_0001_0017.Channel_5.Input <-> Channel 5/Input
//     PlcTask Inputs/GVL_iXlinker.EtherCAT_Master_EPPxxxx.Beckhoff_EPP1xxx.Beckhoff_EPP1xxxEK1122.A_0003_EPP1008_0001_0017.Channel_6.Input <-> Channel 6/Input
//     PlcTask Inputs/GVL_iXlinker.EtherCAT_Master_EPPxxxx.Beckhoff_EPP1xxx.Beckhoff_EPP1xxxEK1122.A_0003_EPP1008_0001_0017.Channel_7.Input <-> Channel 7/Input
//     PlcTask Inputs/GVL_iXlinker.EtherCAT_Master_EPPxxxx.Beckhoff_EPP1xxx.Beckhoff_EPP1xxxEK1122.A_0003_EPP1008_0001_0017.Channel_8.Input <-> Channel 8/Input
//     PlcTask Inputs/GVL_iXlinker.EtherCAT_Master_EPPxxxx.Beckhoff_EPP1xxx.Beckhoff_EPP1xxxEK1122.A_0003_EPP1008_0001_0017.WcState.WcState <-> WcState/WcState
//     PlcTask Inputs/GVL_iXlinker.EtherCAT_Master_EPPxxxx.Beckhoff_EPP1xxx.Beckhoff_EPP1xxxEK1122.A_0003_EPP1008_0001_0017.WcState.InputToggle <-> WcState/InputToggle
//     PlcTask Inputs/GVL_iXlinker.EtherCAT_Master_EPPxxxx.Beckhoff_EPP1xxx.Beckhoff_EPP1xxxEK1122.A_0003_EPP1008_0001_0017.InfoData.State <-> InfoData/State
//   PLC/PLC Instance <-> EtherCAT Master EPPxxxx/Beckhoff EPP1xxx/Beckhoff EPP1xxxEK1122/A_0004(EPP1008-0002-0016)
//     PlcTask Inputs/GVL_iXlinker.EtherCAT_Master_EPPxxxx.Beckhoff_EPP1xxx.Beckhoff_EPP1xxxEK1122.A_0004_EPP1008_0002_0016.Channel_1.Input <-> Channel 1/Input
//     PlcTask Inputs/GVL_iXlinker.EtherCAT_Master_EPPxxxx.Beckhoff_EPP1xxx.Beckhoff_EPP1xxxEK1122.A_0004_EPP1008_0002_0016.Channel_2.Input <-> Channel 2/Input
//     PlcTask Inputs/GVL_iXlinker.EtherCAT_Master_EPPxxxx.Beckhoff_EPP1xxx.Beckhoff_EPP1xxxEK1122.A_0004_EPP1008_0002_0016.Channel_3.Input <-> Channel 3/Input
//     PlcTask Inputs/GVL_iXlinker.EtherCAT_Master_EPPxxxx.Beckhoff_EPP1xxx.Beckhoff_EPP1xxxEK1122.A_0004_EPP1008_0002_0016.Channel_4.Input <-> Channel 4/Input
//     PlcTask Inputs/GVL_iXlinker.EtherCAT_Master_EPPxxxx.Beckhoff_EPP1xxx.Beckhoff_EPP1xxxEK1122.A_0004_EPP1008_0002_0016.Channel_5.Input <-> Channel 5/Input
//     PlcTask Inputs/GVL_iXlinker.EtherCAT_Master_EPPxxxx.Beckhoff_EPP1xxx.Beckhoff_EPP1xxxEK1122.A_0004_EPP1008_0002_0016.Channel_6.Input <-> Channel 6/Input
//     PlcTask Inputs/GVL_iXlinker.EtherCAT_Master_EPPxxxx.Beckhoff_EPP1xxx.Beckhoff_EPP1xxxEK1122.A_0004_EPP1008_0002_0016.Channel_7.Input <-> Channel 7/Input
//     PlcTask Inputs/GVL_iXlinker.EtherCAT_Master_EPPxxxx.Beckhoff_EPP1xxx.Beckhoff_EPP1xxxEK1122.A_0004_EPP1008_0002_0016.Channel_8.Input <-> Channel 8/Input
//     PlcTask Inputs/GVL_iXlinker.EtherCAT_Master_EPPxxxx.Beckhoff_EPP1xxx.Beckhoff_EPP1xxxEK1122.A_0004_EPP1008_0002_0016.WcState.WcState <-> WcState/WcState
//     PlcTask Inputs/GVL_iXlinker.EtherCAT_Master_EPPxxxx.Beckhoff_EPP1xxx.Beckhoff_EPP1xxxEK1122.A_0004_EPP1008_0002_0016.WcState.InputToggle <-> WcState/InputToggle
//     PlcTask Inputs/GVL_iXlinker.EtherCAT_Master_EPPxxxx.Beckhoff_EPP1xxx.Beckhoff_EPP1xxxEK1122.A_0004_EPP1008_0002_0016.InfoData.State <-> InfoData/State
//   PLC/PLC Instance <-> EtherCAT Master EPPxxxx/Beckhoff EPP1xxx/Beckhoff EPP1xxxEK1122/A_0005(EPP1008-0002-0017)
//     PlcTask Inputs/GVL_iXlinker.EtherCAT_Master_EPPxxxx.Beckhoff_EPP1xxx.Beckhoff_EPP1xxxEK1122.A_0005_EPP1008_0002_0017.Channel_1.Input <-> Channel 1/Input
//     PlcTask Inputs/GVL_iXlinker.EtherCAT_Master_EPPxxxx.Beckhoff_EPP1xxx.Beckhoff_EPP1xxxEK1122.A_0005_EPP1008_0002_0017.Channel_2.Input <-> Channel 2/Input
//     PlcTask Inputs/GVL_iXlinker.EtherCAT_Master_EPPxxxx.Beckhoff_EPP1xxx.Beckhoff_EPP1xxxEK1122.A_0005_EPP1008_0002_0017.Channel_3.Input <-> Channel 3/Input
//     PlcTask Inputs/GVL_iXlinker.EtherCAT_Master_EPPxxxx.Beckhoff_EPP1xxx.Beckhoff_EPP1xxxEK1122.A_0005_EPP1008_0002_0017.Channel_4.Input <-> Channel 4/Input
//     PlcTask Inputs/GVL_iXlinker.EtherCAT_Master_EPPxxxx.Beckhoff_EPP1xxx.Beckhoff_EPP1xxxEK1122.A_0005_EPP1008_0002_0017.Channel_5.Input <-> Channel 5/Input
//     PlcTask Inputs/GVL_iXlinker.EtherCAT_Master_EPPxxxx.Beckhoff_EPP1xxx.Beckhoff_EPP1xxxEK1122.A_0005_EPP1008_0002_0017.Channel_6.Input <-> Channel 6/Input
//     PlcTask Inputs/GVL_iXlinker.EtherCAT_Master_EPPxxxx.Beckhoff_EPP1xxx.Beckhoff_EPP1xxxEK1122.A_0005_EPP1008_0002_0017.Channel_7.Input <-> Channel 7/Input
//     PlcTask Inputs/GVL_iXlinker.EtherCAT_Master_EPPxxxx.Beckhoff_EPP1xxx.Beckhoff_EPP1xxxEK1122.A_0005_EPP1008_0002_0017.Channel_8.Input <-> Channel 8/Input
//     PlcTask Inputs/GVL_iXlinker.EtherCAT_Master_EPPxxxx.Beckhoff_EPP1xxx.Beckhoff_EPP1xxxEK1122.A_0005_EPP1008_0002_0017.WcState.WcState <-> WcState/WcState
//     PlcTask Inputs/GVL_iXlinker.EtherCAT_Master_EPPxxxx.Beckhoff_EPP1xxx.Beckhoff_EPP1xxxEK1122.A_0005_EPP1008_0002_0017.WcState.InputToggle <-> WcState/InputToggle
//     PlcTask Inputs/GVL_iXlinker.EtherCAT_Master_EPPxxxx.Beckhoff_EPP1xxx.Beckhoff_EPP1xxxEK1122.A_0005_EPP1008_0002_0017.InfoData.State <-> InfoData/State
//   PLC/PLC Instance <-> EtherCAT Master EPPxxxx/Beckhoff EPP1xxx/Beckhoff EPP1xxxEK1122/A_0006(EPP1008-0022-0016)
//     PlcTask Inputs/GVL_iXlinker.EtherCAT_Master_EPPxxxx.Beckhoff_EPP1xxx.Beckhoff_EPP1xxxEK1122.A_0006_EPP1008_0022_0016.Channel_1.Input <-> Channel 1/Input
//     PlcTask Inputs/GVL_iXlinker.EtherCAT_Master_EPPxxxx.Beckhoff_EPP1xxx.Beckhoff_EPP1xxxEK1122.A_0006_EPP1008_0022_0016.Channel_2.Input <-> Channel 2/Input
//     PlcTask Inputs/GVL_iXlinker.EtherCAT_Master_EPPxxxx.Beckhoff_EPP1xxx.Beckhoff_EPP1xxxEK1122.A_0006_EPP1008_0022_0016.Channel_3.Input <-> Channel 3/Input
//     PlcTask Inputs/GVL_iXlinker.EtherCAT_Master_EPPxxxx.Beckhoff_EPP1xxx.Beckhoff_EPP1xxxEK1122.A_0006_EPP1008_0022_0016.Channel_4.Input <-> Channel 4/Input
//     PlcTask Inputs/GVL_iXlinker.EtherCAT_Master_EPPxxxx.Beckhoff_EPP1xxx.Beckhoff_EPP1xxxEK1122.A_0006_EPP1008_0022_0016.Channel_5.Input <-> Channel 5/Input
//     PlcTask Inputs/GVL_iXlinker.EtherCAT_Master_EPPxxxx.Beckhoff_EPP1xxx.Beckhoff_EPP1xxxEK1122.A_0006_EPP1008_0022_0016.Channel_6.Input <-> Channel 6/Input
//     PlcTask Inputs/GVL_iXlinker.EtherCAT_Master_EPPxxxx.Beckhoff_EPP1xxx.Beckhoff_EPP1xxxEK1122.A_0006_EPP1008_0022_0016.Channel_7.Input <-> Channel 7/Input
//     PlcTask Inputs/GVL_iXlinker.EtherCAT_Master_EPPxxxx.Beckhoff_EPP1xxx.Beckhoff_EPP1xxxEK1122.A_0006_EPP1008_0022_0016.Channel_8.Input <-> Channel 8/Input
//     PlcTask Inputs/GVL_iXlinker.EtherCAT_Master_EPPxxxx.Beckhoff_EPP1xxx.Beckhoff_EPP1xxxEK1122.A_0006_EPP1008_0022_0016.WcState.WcState <-> WcState/WcState
//     PlcTask Inputs/GVL_iXlinker.EtherCAT_Master_EPPxxxx.Beckhoff_EPP1xxx.Beckhoff_EPP1xxxEK1122.A_0006_EPP1008_0022_0016.WcState.InputToggle <-> WcState/InputToggle
//     PlcTask Inputs/GVL_iXlinker.EtherCAT_Master_EPPxxxx.Beckhoff_EPP1xxx.Beckhoff_EPP1xxxEK1122.A_0006_EPP1008_0022_0016.InfoData.State <-> InfoData/State
//   PLC/PLC Instance <-> EtherCAT Master EPPxxxx/Beckhoff EPP1xxx/Beckhoff EPP1xxxEK1122/A_0007(EPP1018-0001-0016)
//     PlcTask Inputs/GVL_iXlinker.EtherCAT_Master_EPPxxxx.Beckhoff_EPP1xxx.Beckhoff_EPP1xxxEK1122.A_0007_EPP1018_0001_0016.Channel_1.Input <-> Channel 1/Input
//     PlcTask Inputs/GVL_iXlinker.EtherCAT_Master_EPPxxxx.Beckhoff_EPP1xxx.Beckhoff_EPP1xxxEK1122.A_0007_EPP1018_0001_0016.Channel_2.Input <-> Channel 2/Input
//     PlcTask Inputs/GVL_iXlinker.EtherCAT_Master_EPPxxxx.Beckhoff_EPP1xxx.Beckhoff_EPP1xxxEK1122.A_0007_EPP1018_0001_0016.Channel_3.Input <-> Channel 3/Input
//     PlcTask Inputs/GVL_iXlinker.EtherCAT_Master_EPPxxxx.Beckhoff_EPP1xxx.Beckhoff_EPP1xxxEK1122.A_0007_EPP1018_0001_0016.Channel_4.Input <-> Channel 4/Input
//     PlcTask Inputs/GVL_iXlinker.EtherCAT_Master_EPPxxxx.Beckhoff_EPP1xxx.Beckhoff_EPP1xxxEK1122.A_0007_EPP1018_0001_0016.Channel_5.Input <-> Channel 5/Input
//     PlcTask Inputs/GVL_iXlinker.EtherCAT_Master_EPPxxxx.Beckhoff_EPP1xxx.Beckhoff_EPP1xxxEK1122.A_0007_EPP1018_0001_0016.Channel_6.Input <-> Channel 6/Input
//     PlcTask Inputs/GVL_iXlinker.EtherCAT_Master_EPPxxxx.Beckhoff_EPP1xxx.Beckhoff_EPP1xxxEK1122.A_0007_EPP1018_0001_0016.Channel_7.Input <-> Channel 7/Input
//     PlcTask Inputs/GVL_iXlinker.EtherCAT_Master_EPPxxxx.Beckhoff_EPP1xxx.Beckhoff_EPP1xxxEK1122.A_0007_EPP1018_0001_0016.Channel_8.Input <-> Channel 8/Input
//     PlcTask Inputs/GVL_iXlinker.EtherCAT_Master_EPPxxxx.Beckhoff_EPP1xxx.Beckhoff_EPP1xxxEK1122.A_0007_EPP1018_0001_0016.WcState.WcState <-> WcState/WcState
//     PlcTask Inputs/GVL_iXlinker.EtherCAT_Master_EPPxxxx.Beckhoff_EPP1xxx.Beckhoff_EPP1xxxEK1122.A_0007_EPP1018_0001_0016.WcState.InputToggle <-> WcState/InputToggle
//     PlcTask Inputs/GVL_iXlinker.EtherCAT_Master_EPPxxxx.Beckhoff_EPP1xxx.Beckhoff_EPP1xxxEK1122.A_0007_EPP1018_0001_0016.InfoData.State <-> InfoData/State
//   PLC/PLC Instance <-> EtherCAT Master EPPxxxx/Beckhoff EPP1xxx/Beckhoff EPP1xxxEK1122/A_0008(EPP1018-0001-0017)
//     PlcTask Inputs/GVL_iXlinker.EtherCAT_Master_EPPxxxx.Beckhoff_EPP1xxx.Beckhoff_EPP1xxxEK1122.A_0008_EPP1018_0001_0017.Channel_1.Input <-> Channel 1/Input
//     PlcTask Inputs/GVL_iXlinker.EtherCAT_Master_EPPxxxx.Beckhoff_EPP1xxx.Beckhoff_EPP1xxxEK1122.A_0008_EPP1018_0001_0017.Channel_2.Input <-> Channel 2/Input
//     PlcTask Inputs/GVL_iXlinker.EtherCAT_Master_EPPxxxx.Beckhoff_EPP1xxx.Beckhoff_EPP1xxxEK1122.A_0008_EPP1018_0001_0017.Channel_3.Input <-> Channel 3/Input
//     PlcTask Inputs/GVL_iXlinker.EtherCAT_Master_EPPxxxx.Beckhoff_EPP1xxx.Beckhoff_EPP1xxxEK1122.A_0008_EPP1018_0001_0017.Channel_4.Input <-> Channel 4/Input
//     PlcTask Inputs/GVL_iXlinker.EtherCAT_Master_EPPxxxx.Beckhoff_EPP1xxx.Beckhoff_EPP1xxxEK1122.A_0008_EPP1018_0001_0017.Channel_5.Input <-> Channel 5/Input
//     PlcTask Inputs/GVL_iXlinker.EtherCAT_Master_EPPxxxx.Beckhoff_EPP1xxx.Beckhoff_EPP1xxxEK1122.A_0008_EPP1018_0001_0017.Channel_6.Input <-> Channel 6/Input
//     PlcTask Inputs/GVL_iXlinker.EtherCAT_Master_EPPxxxx.Beckhoff_EPP1xxx.Beckhoff_EPP1xxxEK1122.A_0008_EPP1018_0001_0017.Channel_7.Input <-> Channel 7/Input
//     PlcTask Inputs/GVL_iXlinker.EtherCAT_Master_EPPxxxx.Beckhoff_EPP1xxx.Beckhoff_EPP1xxxEK1122.A_0008_EPP1018_0001_0017.Channel_8.Input <-> Channel 8/Input
//     PlcTask Inputs/GVL_iXlinker.EtherCAT_Master_EPPxxxx.Beckhoff_EPP1xxx.Beckhoff_EPP1xxxEK1122.A_0008_EPP1018_0001_0017.WcState.WcState <-> WcState/WcState
//     PlcTask Inputs/GVL_iXlinker.EtherCAT_Master_EPPxxxx.Beckhoff_EPP1xxx.Beckhoff_EPP1xxxEK1122.A_0008_EPP1018_0001_0017.WcState.InputToggle <-> WcState/InputToggle
//     PlcTask Inputs/GVL_iXlinker.EtherCAT_Master_EPPxxxx.Beckhoff_EPP1xxx.Beckhoff_EPP1xxxEK1122.A_0008_EPP1018_0001_0017.InfoData.State <-> InfoData/State
//   PLC/PLC Instance <-> EtherCAT Master EPPxxxx/Beckhoff EPP1xxx/Beckhoff EPP1xxxEK1122/A_0009(EPP1018-0002-0016)
//     PlcTask Inputs/GVL_iXlinker.EtherCAT_Master_EPPxxxx.Beckhoff_EPP1xxx.Beckhoff_EPP1xxxEK1122.A_0009_EPP1018_0002_0016.Channel_1.Input <-> Channel 1/Input
//     PlcTask Inputs/GVL_iXlinker.EtherCAT_Master_EPPxxxx.Beckhoff_EPP1xxx.Beckhoff_EPP1xxxEK1122.A_0009_EPP1018_0002_0016.Channel_2.Input <-> Channel 2/Input
//     PlcTask Inputs/GVL_iXlinker.EtherCAT_Master_EPPxxxx.Beckhoff_EPP1xxx.Beckhoff_EPP1xxxEK1122.A_0009_EPP1018_0002_0016.Channel_3.Input <-> Channel 3/Input
//     PlcTask Inputs/GVL_iXlinker.EtherCAT_Master_EPPxxxx.Beckhoff_EPP1xxx.Beckhoff_EPP1xxxEK1122.A_0009_EPP1018_0002_0016.Channel_4.Input <-> Channel 4/Input
//     PlcTask Inputs/GVL_iXlinker.EtherCAT_Master_EPPxxxx.Beckhoff_EPP1xxx.Beckhoff_EPP1xxxEK1122.A_0009_EPP1018_0002_0016.Channel_5.Input <-> Channel 5/Input
//     PlcTask Inputs/GVL_iXlinker.EtherCAT_Master_EPPxxxx.Beckhoff_EPP1xxx.Beckhoff_EPP1xxxEK1122.A_0009_EPP1018_0002_0016.Channel_6.Input <-> Channel 6/Input
//     PlcTask Inputs/GVL_iXlinker.EtherCAT_Master_EPPxxxx.Beckhoff_EPP1xxx.Beckhoff_EPP1xxxEK1122.A_0009_EPP1018_0002_0016.Channel_7.Input <-> Channel 7/Input
//     PlcTask Inputs/GVL_iXlinker.EtherCAT_Master_EPPxxxx.Beckhoff_EPP1xxx.Beckhoff_EPP1xxxEK1122.A_0009_EPP1018_0002_0016.Channel_8.Input <-> Channel 8/Input
//     PlcTask Inputs/GVL_iXlinker.EtherCAT_Master_EPPxxxx.Beckhoff_EPP1xxx.Beckhoff_EPP1xxxEK1122.A_0009_EPP1018_0002_0016.WcState.WcState <-> WcState/WcState
//     PlcTask Inputs/GVL_iXlinker.EtherCAT_Master_EPPxxxx.Beckhoff_EPP1xxx.Beckhoff_EPP1xxxEK1122.A_0009_EPP1018_0002_0016.WcState.InputToggle <-> WcState/InputToggle
//     PlcTask Inputs/GVL_iXlinker.EtherCAT_Master_EPPxxxx.Beckhoff_EPP1xxx.Beckhoff_EPP1xxxEK1122.A_0009_EPP1018_0002_0016.InfoData.State <-> InfoData/State
//   PLC/PLC Instance <-> EtherCAT Master EPPxxxx/Beckhoff EPP1xxx/Beckhoff EPP1xxxEK1122/A_0010(EPP1018-0002-0017)
//     PlcTask Inputs/GVL_iXlinker.EtherCAT_Master_EPPxxxx.Beckhoff_EPP1xxx.Beckhoff_EPP1xxxEK1122.A_0010_EPP1018_0002_0017.Channel_1.Input <-> Channel 1/Input
//     PlcTask Inputs/GVL_iXlinker.EtherCAT_Master_EPPxxxx.Beckhoff_EPP1xxx.Beckhoff_EPP1xxxEK1122.A_0010_EPP1018_0002_0017.Channel_2.Input <-> Channel 2/Input
//     PlcTask Inputs/GVL_iXlinker.EtherCAT_Master_EPPxxxx.Beckhoff_EPP1xxx.Beckhoff_EPP1xxxEK1122.A_0010_EPP1018_0002_0017.Channel_3.Input <-> Channel 3/Input
//     PlcTask Inputs/GVL_iXlinker.EtherCAT_Master_EPPxxxx.Beckhoff_EPP1xxx.Beckhoff_EPP1xxxEK1122.A_0010_EPP1018_0002_0017.Channel_4.Input <-> Channel 4/Input
//     PlcTask Inputs/GVL_iXlinker.EtherCAT_Master_EPPxxxx.Beckhoff_EPP1xxx.Beckhoff_EPP1xxxEK1122.A_0010_EPP1018_0002_0017.Channel_5.Input <-> Channel 5/Input
//     PlcTask Inputs/GVL_iXlinker.EtherCAT_Master_EPPxxxx.Beckhoff_EPP1xxx.Beckhoff_EPP1xxxEK1122.A_0010_EPP1018_0002_0017.Channel_6.Input <-> Channel 6/Input
//     PlcTask Inputs/GVL_iXlinker.EtherCAT_Master_EPPxxxx.Beckhoff_EPP1xxx.Beckhoff_EPP1xxxEK1122.A_0010_EPP1018_0002_0017.Channel_7.Input <-> Channel 7/Input
//     PlcTask Inputs/GVL_iXlinker.EtherCAT_Master_EPPxxxx.Beckhoff_EPP1xxx.Beckhoff_EPP1xxxEK1122.A_0010_EPP1018_0002_0017.Channel_8.Input <-> Channel 8/Input
//     PlcTask Inputs/GVL_iXlinker.EtherCAT_Master_EPPxxxx.Beckhoff_EPP1xxx.Beckhoff_EPP1xxxEK1122.A_0010_EPP1018_0002_0017.WcState.WcState <-> WcState/WcState
//     PlcTask Inputs/GVL_iXlinker.EtherCAT_Master_EPPxxxx.Beckhoff_EPP1xxx.Beckhoff_EPP1xxxEK1122.A_0010_EPP1018_0002_0017.WcState.InputToggle <-> WcState/InputToggle
//     PlcTask Inputs/GVL_iXlinker.EtherCAT_Master_EPPxxxx.Beckhoff_EPP1xxx.Beckhoff_EPP1xxxEK1122.A_0010_EPP1018_0002_0017.InfoData.State <-> InfoData/State
//   PLC/PLC Instance <-> EtherCAT Master EPPxxxx/Beckhoff EPP1xxx/Beckhoff EPP1xxxEK1122/A_0011(EPP1111-0000-0016)
//     PlcTask Inputs/GVL_iXlinker.EtherCAT_Master_EPPxxxx.Beckhoff_EPP1xxx.Beckhoff_EPP1xxxEK1122.A_0011_EPP1111_0000_0016.ID_Inputs.ID <-> ID Inputs /ID
//     PlcTask Inputs/GVL_iXlinker.EtherCAT_Master_EPPxxxx.Beckhoff_EPP1xxx.Beckhoff_EPP1xxxEK1122.A_0011_EPP1111_0000_0016.WcState.WcState <-> WcState/WcState
//     PlcTask Inputs/GVL_iXlinker.EtherCAT_Master_EPPxxxx.Beckhoff_EPP1xxx.Beckhoff_EPP1xxxEK1122.A_0011_EPP1111_0000_0016.WcState.InputToggle <-> WcState/InputToggle
//     PlcTask Inputs/GVL_iXlinker.EtherCAT_Master_EPPxxxx.Beckhoff_EPP1xxx.Beckhoff_EPP1xxxEK1122.A_0011_EPP1111_0000_0016.InfoData.AdsAddr <-> InfoData/AdsAddr
//     PlcTask Inputs/GVL_iXlinker.EtherCAT_Master_EPPxxxx.Beckhoff_EPP1xxx.Beckhoff_EPP1xxxEK1122.A_0011_EPP1111_0000_0016.InfoData.State <-> InfoData/State
//   PLC/PLC Instance <-> EtherCAT Master EPPxxxx/Beckhoff EPP1xxx/Beckhoff EPP1xxxEK1122/A_0012(EPP1111-0000-0017)
//     PlcTask Inputs/GVL_iXlinker.EtherCAT_Master_EPPxxxx.Beckhoff_EPP1xxx.Beckhoff_EPP1xxxEK1122.A_0012_EPP1111_0000_0017.ID_Inputs.ID <-> ID Inputs/ID
//     PlcTask Inputs/GVL_iXlinker.EtherCAT_Master_EPPxxxx.Beckhoff_EPP1xxx.Beckhoff_EPP1xxxEK1122.A_0012_EPP1111_0000_0017.WcState.WcState <-> WcState/WcState
//     PlcTask Inputs/GVL_iXlinker.EtherCAT_Master_EPPxxxx.Beckhoff_EPP1xxx.Beckhoff_EPP1xxxEK1122.A_0012_EPP1111_0000_0017.WcState.InputToggle <-> WcState/InputToggle
//     PlcTask Inputs/GVL_iXlinker.EtherCAT_Master_EPPxxxx.Beckhoff_EPP1xxx.Beckhoff_EPP1xxxEK1122.A_0012_EPP1111_0000_0017.InfoData.AdsAddr <-> InfoData/AdsAddr
//     PlcTask Inputs/GVL_iXlinker.EtherCAT_Master_EPPxxxx.Beckhoff_EPP1xxx.Beckhoff_EPP1xxxEK1122.A_0012_EPP1111_0000_0017.InfoData.State <-> InfoData/State
//   PLC/PLC Instance <-> EtherCAT Master EPPxxxx/Beckhoff EPP1xxx/Beckhoff EPP1xxxEK1122/A_0013(EPP1111-0000-0018)
//     PlcTask Inputs/GVL_iXlinker.EtherCAT_Master_EPPxxxx.Beckhoff_EPP1xxx.Beckhoff_EPP1xxxEK1122.A_0013_EPP1111_0000_0018.ID_Inputs.ID <-> ID Inputs/ID
//     PlcTask Inputs/GVL_iXlinker.EtherCAT_Master_EPPxxxx.Beckhoff_EPP1xxx.Beckhoff_EPP1xxxEK1122.A_0013_EPP1111_0000_0018.WcState.WcState <-> WcState/WcState
//     PlcTask Inputs/GVL_iXlinker.EtherCAT_Master_EPPxxxx.Beckhoff_EPP1xxx.Beckhoff_EPP1xxxEK1122.A_0013_EPP1111_0000_0018.WcState.InputToggle <-> WcState/InputToggle
//     PlcTask Inputs/GVL_iXlinker.EtherCAT_Master_EPPxxxx.Beckhoff_EPP1xxx.Beckhoff_EPP1xxxEK1122.A_0013_EPP1111_0000_0018.InfoData.AdsAddr <-> InfoData/AdsAddr
//     PlcTask Inputs/GVL_iXlinker.EtherCAT_Master_EPPxxxx.Beckhoff_EPP1xxx.Beckhoff_EPP1xxxEK1122.A_0013_EPP1111_0000_0018.InfoData.State <-> InfoData/State
//   PLC/PLC Instance <-> EtherCAT Master EPPxxxx/Beckhoff EPP1xxx/Beckhoff EPP1xxxEK1122/A_0014(EPP1258-0001-0016)
//     PlcTask Inputs/GVL_iXlinker.EtherCAT_Master_EPPxxxx.Beckhoff_EPP1xxx.Beckhoff_EPP1xxxEK1122.A_0014_EPP1258_0001_0016.Channel_1.Input <-> Channel 1/Input
//     PlcTask Inputs/GVL_iXlinker.EtherCAT_Master_EPPxxxx.Beckhoff_EPP1xxx.Beckhoff_EPP1xxxEK1122.A_0014_EPP1258_0001_0016.Channel_2.Input <-> Channel 2/Input
//     PlcTask Inputs/GVL_iXlinker.EtherCAT_Master_EPPxxxx.Beckhoff_EPP1xxx.Beckhoff_EPP1xxxEK1122.A_0014_EPP1258_0001_0016.Channel_3.Input <-> Channel 3/Input
//     PlcTask Inputs/GVL_iXlinker.EtherCAT_Master_EPPxxxx.Beckhoff_EPP1xxx.Beckhoff_EPP1xxxEK1122.A_0014_EPP1258_0001_0016.Channel_4.Input <-> Channel 4/Input
//     PlcTask Inputs/GVL_iXlinker.EtherCAT_Master_EPPxxxx.Beckhoff_EPP1xxx.Beckhoff_EPP1xxxEK1122.A_0014_EPP1258_0001_0016.Channel_5.Input <-> Channel 5/Input
//     PlcTask Inputs/GVL_iXlinker.EtherCAT_Master_EPPxxxx.Beckhoff_EPP1xxx.Beckhoff_EPP1xxxEK1122.A_0014_EPP1258_0001_0016.Channel_6.Input <-> Channel 6/Input
//     PlcTask Inputs/GVL_iXlinker.EtherCAT_Master_EPPxxxx.Beckhoff_EPP1xxx.Beckhoff_EPP1xxxEK1122.A_0014_EPP1258_0001_0016.Channel_7.Input <-> Channel 7/Input
//     PlcTask Inputs/GVL_iXlinker.EtherCAT_Master_EPPxxxx.Beckhoff_EPP1xxx.Beckhoff_EPP1xxxEK1122.A_0014_EPP1258_0001_0016.Channel_8.Input <-> Channel 8/Input
//     PlcTask Inputs/GVL_iXlinker.EtherCAT_Master_EPPxxxx.Beckhoff_EPP1xxx.Beckhoff_EPP1xxxEK1122.A_0014_EPP1258_0001_0016.Latch.Status0 <-> Latch/Status0
//     PlcTask Inputs/GVL_iXlinker.EtherCAT_Master_EPPxxxx.Beckhoff_EPP1xxx.Beckhoff_EPP1xxxEK1122.A_0014_EPP1258_0001_0016.Latch.Status1 <-> Latch/Status1
//     PlcTask Inputs/GVL_iXlinker.EtherCAT_Master_EPPxxxx.Beckhoff_EPP1xxx.Beckhoff_EPP1xxxEK1122.A_0014_EPP1258_0001_0016.Latch.LatchPos0 <-> Latch/LatchPos0
//     PlcTask Inputs/GVL_iXlinker.EtherCAT_Master_EPPxxxx.Beckhoff_EPP1xxx.Beckhoff_EPP1xxxEK1122.A_0014_EPP1258_0001_0016.Latch.LatchPos1 <-> Latch/LatchPos1
//     PlcTask Inputs/GVL_iXlinker.EtherCAT_Master_EPPxxxx.Beckhoff_EPP1xxx.Beckhoff_EPP1xxxEK1122.A_0014_EPP1258_0001_0016.Latch.LatchNeg0 <-> Latch/LatchNeg0
//     PlcTask Inputs/GVL_iXlinker.EtherCAT_Master_EPPxxxx.Beckhoff_EPP1xxx.Beckhoff_EPP1xxxEK1122.A_0014_EPP1258_0001_0016.Latch.LatchNeg1 <-> Latch/LatchNeg1
//     PlcTask Inputs/GVL_iXlinker.EtherCAT_Master_EPPxxxx.Beckhoff_EPP1xxx.Beckhoff_EPP1xxxEK1122.A_0014_EPP1258_0001_0016.WcState.WcState0 <-> WcState/WcState0
//     PlcTask Inputs/GVL_iXlinker.EtherCAT_Master_EPPxxxx.Beckhoff_EPP1xxx.Beckhoff_EPP1xxxEK1122.A_0014_EPP1258_0001_0016.WcState.WcState1 <-> WcState/WcState1
//     PlcTask Inputs/GVL_iXlinker.EtherCAT_Master_EPPxxxx.Beckhoff_EPP1xxx.Beckhoff_EPP1xxxEK1122.A_0014_EPP1258_0001_0016.WcState.InputToggle0 <-> WcState/InputToggle0
//     PlcTask Inputs/GVL_iXlinker.EtherCAT_Master_EPPxxxx.Beckhoff_EPP1xxx.Beckhoff_EPP1xxxEK1122.A_0014_EPP1258_0001_0016.WcState.InputToggle1 <-> WcState/InputToggle1
//     PlcTask Inputs/GVL_iXlinker.EtherCAT_Master_EPPxxxx.Beckhoff_EPP1xxx.Beckhoff_EPP1xxxEK1122.A_0014_EPP1258_0001_0016.InfoData.DcOutputShift <-> InfoData/DcOutputShift
//     PlcTask Inputs/GVL_iXlinker.EtherCAT_Master_EPPxxxx.Beckhoff_EPP1xxx.Beckhoff_EPP1xxxEK1122.A_0014_EPP1258_0001_0016.InfoData.DcInputShift <-> InfoData/DcInputShift
//     PlcTask Inputs/GVL_iXlinker.EtherCAT_Master_EPPxxxx.Beckhoff_EPP1xxx.Beckhoff_EPP1xxxEK1122.A_0014_EPP1258_0001_0016.InfoData.State <-> InfoData/State
//   PLC/PLC Instance <-> EtherCAT Master EPPxxxx/Beckhoff EPP1xxx/Beckhoff EPP1xxxEK1122/A_0015(EPP1258-0001-0017)
//     PlcTask Inputs/GVL_iXlinker.EtherCAT_Master_EPPxxxx.Beckhoff_EPP1xxx.Beckhoff_EPP1xxxEK1122.A_0015_EPP1258_0001_0017.Channel_1.Input <-> Channel 1/Input
//     PlcTask Inputs/GVL_iXlinker.EtherCAT_Master_EPPxxxx.Beckhoff_EPP1xxx.Beckhoff_EPP1xxxEK1122.A_0015_EPP1258_0001_0017.Channel_2.Input <-> Channel 2/Input
//     PlcTask Inputs/GVL_iXlinker.EtherCAT_Master_EPPxxxx.Beckhoff_EPP1xxx.Beckhoff_EPP1xxxEK1122.A_0015_EPP1258_0001_0017.Channel_3.Input <-> Channel 3/Input
//     PlcTask Inputs/GVL_iXlinker.EtherCAT_Master_EPPxxxx.Beckhoff_EPP1xxx.Beckhoff_EPP1xxxEK1122.A_0015_EPP1258_0001_0017.Channel_4.Input <-> Channel 4/Input
//     PlcTask Inputs/GVL_iXlinker.EtherCAT_Master_EPPxxxx.Beckhoff_EPP1xxx.Beckhoff_EPP1xxxEK1122.A_0015_EPP1258_0001_0017.Channel_5.Input <-> Channel 5/Input
//     PlcTask Inputs/GVL_iXlinker.EtherCAT_Master_EPPxxxx.Beckhoff_EPP1xxx.Beckhoff_EPP1xxxEK1122.A_0015_EPP1258_0001_0017.Channel_6.Input <-> Channel 6/Input
//     PlcTask Inputs/GVL_iXlinker.EtherCAT_Master_EPPxxxx.Beckhoff_EPP1xxx.Beckhoff_EPP1xxxEK1122.A_0015_EPP1258_0001_0017.Channel_7.Input <-> Channel 7/Input
//     PlcTask Inputs/GVL_iXlinker.EtherCAT_Master_EPPxxxx.Beckhoff_EPP1xxx.Beckhoff_EPP1xxxEK1122.A_0015_EPP1258_0001_0017.Channel_8.Input <-> Channel 8/Input
//     PlcTask Inputs/GVL_iXlinker.EtherCAT_Master_EPPxxxx.Beckhoff_EPP1xxx.Beckhoff_EPP1xxxEK1122.A_0015_EPP1258_0001_0017.Latch.Status0 <-> Latch/Status0
//     PlcTask Inputs/GVL_iXlinker.EtherCAT_Master_EPPxxxx.Beckhoff_EPP1xxx.Beckhoff_EPP1xxxEK1122.A_0015_EPP1258_0001_0017.Latch.Status1 <-> Latch/Status1
//     PlcTask Inputs/GVL_iXlinker.EtherCAT_Master_EPPxxxx.Beckhoff_EPP1xxx.Beckhoff_EPP1xxxEK1122.A_0015_EPP1258_0001_0017.Latch.LatchPos0 <-> Latch/LatchPos0
//     PlcTask Inputs/GVL_iXlinker.EtherCAT_Master_EPPxxxx.Beckhoff_EPP1xxx.Beckhoff_EPP1xxxEK1122.A_0015_EPP1258_0001_0017.Latch.LatchPos1 <-> Latch/LatchPos1
//     PlcTask Inputs/GVL_iXlinker.EtherCAT_Master_EPPxxxx.Beckhoff_EPP1xxx.Beckhoff_EPP1xxxEK1122.A_0015_EPP1258_0001_0017.Latch.LatchNeg0 <-> Latch/LatchNeg0
//     PlcTask Inputs/GVL_iXlinker.EtherCAT_Master_EPPxxxx.Beckhoff_EPP1xxx.Beckhoff_EPP1xxxEK1122.A_0015_EPP1258_0001_0017.Latch.LatchNeg1 <-> Latch/LatchNeg1
//     PlcTask Inputs/GVL_iXlinker.EtherCAT_Master_EPPxxxx.Beckhoff_EPP1xxx.Beckhoff_EPP1xxxEK1122.A_0015_EPP1258_0001_0017.WcState.WcState0 <-> WcState/WcState0
//     PlcTask Inputs/GVL_iXlinker.EtherCAT_Master_EPPxxxx.Beckhoff_EPP1xxx.Beckhoff_EPP1xxxEK1122.A_0015_EPP1258_0001_0017.WcState.WcState1 <-> WcState/WcState1
//     PlcTask Inputs/GVL_iXlinker.EtherCAT_Master_EPPxxxx.Beckhoff_EPP1xxx.Beckhoff_EPP1xxxEK1122.A_0015_EPP1258_0001_0017.WcState.InputToggle0 <-> WcState/InputToggle0
//     PlcTask Inputs/GVL_iXlinker.EtherCAT_Master_EPPxxxx.Beckhoff_EPP1xxx.Beckhoff_EPP1xxxEK1122.A_0015_EPP1258_0001_0017.WcState.InputToggle1 <-> WcState/InputToggle1
//     PlcTask Inputs/GVL_iXlinker.EtherCAT_Master_EPPxxxx.Beckhoff_EPP1xxx.Beckhoff_EPP1xxxEK1122.A_0015_EPP1258_0001_0017.InfoData.DcOutputShift <-> InfoData/DcOutputShift
//     PlcTask Inputs/GVL_iXlinker.EtherCAT_Master_EPPxxxx.Beckhoff_EPP1xxx.Beckhoff_EPP1xxxEK1122.A_0015_EPP1258_0001_0017.InfoData.DcInputShift <-> InfoData/DcInputShift
//     PlcTask Inputs/GVL_iXlinker.EtherCAT_Master_EPPxxxx.Beckhoff_EPP1xxx.Beckhoff_EPP1xxxEK1122.A_0015_EPP1258_0001_0017.InfoData.State <-> InfoData/State
//   PLC/PLC Instance <-> EtherCAT Master EPPxxxx/Beckhoff EPP1xxx/Beckhoff EPP1xxxEK1122/A_0016(EPP1258-0002-0016)
//     PlcTask Inputs/GVL_iXlinker.EtherCAT_Master_EPPxxxx.Beckhoff_EPP1xxx.Beckhoff_EPP1xxxEK1122.A_0016_EPP1258_0002_0016.Channel_1.Input <-> Channel 1/Input
//     PlcTask Inputs/GVL_iXlinker.EtherCAT_Master_EPPxxxx.Beckhoff_EPP1xxx.Beckhoff_EPP1xxxEK1122.A_0016_EPP1258_0002_0016.Channel_2.Input <-> Channel 2/Input
//     PlcTask Inputs/GVL_iXlinker.EtherCAT_Master_EPPxxxx.Beckhoff_EPP1xxx.Beckhoff_EPP1xxxEK1122.A_0016_EPP1258_0002_0016.Channel_3.Input <-> Channel 3/Input
//     PlcTask Inputs/GVL_iXlinker.EtherCAT_Master_EPPxxxx.Beckhoff_EPP1xxx.Beckhoff_EPP1xxxEK1122.A_0016_EPP1258_0002_0016.Channel_4.Input <-> Channel 4/Input
//     PlcTask Inputs/GVL_iXlinker.EtherCAT_Master_EPPxxxx.Beckhoff_EPP1xxx.Beckhoff_EPP1xxxEK1122.A_0016_EPP1258_0002_0016.Channel_5.Input <-> Channel 5/Input
//     PlcTask Inputs/GVL_iXlinker.EtherCAT_Master_EPPxxxx.Beckhoff_EPP1xxx.Beckhoff_EPP1xxxEK1122.A_0016_EPP1258_0002_0016.Channel_6.Input <-> Channel 6/Input
//     PlcTask Inputs/GVL_iXlinker.EtherCAT_Master_EPPxxxx.Beckhoff_EPP1xxx.Beckhoff_EPP1xxxEK1122.A_0016_EPP1258_0002_0016.Channel_7.Input <-> Channel 7/Input
//     PlcTask Inputs/GVL_iXlinker.EtherCAT_Master_EPPxxxx.Beckhoff_EPP1xxx.Beckhoff_EPP1xxxEK1122.A_0016_EPP1258_0002_0016.Channel_8.Input <-> Channel 8/Input
//     PlcTask Inputs/GVL_iXlinker.EtherCAT_Master_EPPxxxx.Beckhoff_EPP1xxx.Beckhoff_EPP1xxxEK1122.A_0016_EPP1258_0002_0016.Latch.Status0 <-> Latch/Status0
//     PlcTask Inputs/GVL_iXlinker.EtherCAT_Master_EPPxxxx.Beckhoff_EPP1xxx.Beckhoff_EPP1xxxEK1122.A_0016_EPP1258_0002_0016.Latch.Status1 <-> Latch/Status1
//     PlcTask Inputs/GVL_iXlinker.EtherCAT_Master_EPPxxxx.Beckhoff_EPP1xxx.Beckhoff_EPP1xxxEK1122.A_0016_EPP1258_0002_0016.Latch.LatchPos0 <-> Latch/LatchPos0
//     PlcTask Inputs/GVL_iXlinker.EtherCAT_Master_EPPxxxx.Beckhoff_EPP1xxx.Beckhoff_EPP1xxxEK1122.A_0016_EPP1258_0002_0016.Latch.LatchPos1 <-> Latch/LatchPos1
//     PlcTask Inputs/GVL_iXlinker.EtherCAT_Master_EPPxxxx.Beckhoff_EPP1xxx.Beckhoff_EPP1xxxEK1122.A_0016_EPP1258_0002_0016.Latch.LatchNeg0 <-> Latch/LatchNeg0
//     PlcTask Inputs/GVL_iXlinker.EtherCAT_Master_EPPxxxx.Beckhoff_EPP1xxx.Beckhoff_EPP1xxxEK1122.A_0016_EPP1258_0002_0016.Latch.LatchNeg1 <-> Latch/LatchNeg1
//     PlcTask Inputs/GVL_iXlinker.EtherCAT_Master_EPPxxxx.Beckhoff_EPP1xxx.Beckhoff_EPP1xxxEK1122.A_0016_EPP1258_0002_0016.WcState.WcState0 <-> WcState/WcState0
//     PlcTask Inputs/GVL_iXlinker.EtherCAT_Master_EPPxxxx.Beckhoff_EPP1xxx.Beckhoff_EPP1xxxEK1122.A_0016_EPP1258_0002_0016.WcState.WcState1 <-> WcState/WcState1
//     PlcTask Inputs/GVL_iXlinker.EtherCAT_Master_EPPxxxx.Beckhoff_EPP1xxx.Beckhoff_EPP1xxxEK1122.A_0016_EPP1258_0002_0016.WcState.InputToggle0 <-> WcState/InputToggle0
//     PlcTask Inputs/GVL_iXlinker.EtherCAT_Master_EPPxxxx.Beckhoff_EPP1xxx.Beckhoff_EPP1xxxEK1122.A_0016_EPP1258_0002_0016.WcState.InputToggle1 <-> WcState/InputToggle1
//     PlcTask Inputs/GVL_iXlinker.EtherCAT_Master_EPPxxxx.Beckhoff_EPP1xxx.Beckhoff_EPP1xxxEK1122.A_0016_EPP1258_0002_0016.InfoData.DcOutputShift <-> InfoData/DcOutputShift
//     PlcTask Inputs/GVL_iXlinker.EtherCAT_Master_EPPxxxx.Beckhoff_EPP1xxx.Beckhoff_EPP1xxxEK1122.A_0016_EPP1258_0002_0016.InfoData.DcInputShift <-> InfoData/DcInputShift
//     PlcTask Inputs/GVL_iXlinker.EtherCAT_Master_EPPxxxx.Beckhoff_EPP1xxx.Beckhoff_EPP1xxxEK1122.A_0016_EPP1258_0002_0016.InfoData.State <-> InfoData/State
//   PLC/PLC Instance <-> EtherCAT Master EPPxxxx/Beckhoff EPP1xxx/Beckhoff EPP1xxxEK1122/A_0017(EPP1258-0002-0017)
//     PlcTask Inputs/GVL_iXlinker.EtherCAT_Master_EPPxxxx.Beckhoff_EPP1xxx.Beckhoff_EPP1xxxEK1122.A_0017_EPP1258_0002_0017.Channel_1.Input <-> Channel 1/Input
//     PlcTask Inputs/GVL_iXlinker.EtherCAT_Master_EPPxxxx.Beckhoff_EPP1xxx.Beckhoff_EPP1xxxEK1122.A_0017_EPP1258_0002_0017.Channel_2.Input <-> Channel 2/Input
//     PlcTask Inputs/GVL_iXlinker.EtherCAT_Master_EPPxxxx.Beckhoff_EPP1xxx.Beckhoff_EPP1xxxEK1122.A_0017_EPP1258_0002_0017.Channel_3.Input <-> Channel 3/Input
//     PlcTask Inputs/GVL_iXlinker.EtherCAT_Master_EPPxxxx.Beckhoff_EPP1xxx.Beckhoff_EPP1xxxEK1122.A_0017_EPP1258_0002_0017.Channel_4.Input <-> Channel 4/Input
//     PlcTask Inputs/GVL_iXlinker.EtherCAT_Master_EPPxxxx.Beckhoff_EPP1xxx.Beckhoff_EPP1xxxEK1122.A_0017_EPP1258_0002_0017.Channel_5.Input <-> Channel 5/Input
//     PlcTask Inputs/GVL_iXlinker.EtherCAT_Master_EPPxxxx.Beckhoff_EPP1xxx.Beckhoff_EPP1xxxEK1122.A_0017_EPP1258_0002_0017.Channel_6.Input <-> Channel 6/Input
//     PlcTask Inputs/GVL_iXlinker.EtherCAT_Master_EPPxxxx.Beckhoff_EPP1xxx.Beckhoff_EPP1xxxEK1122.A_0017_EPP1258_0002_0017.Channel_7.Input <-> Channel 7/Input
//     PlcTask Inputs/GVL_iXlinker.EtherCAT_Master_EPPxxxx.Beckhoff_EPP1xxx.Beckhoff_EPP1xxxEK1122.A_0017_EPP1258_0002_0017.Channel_8.Input <-> Channel 8/Input
//     PlcTask Inputs/GVL_iXlinker.EtherCAT_Master_EPPxxxx.Beckhoff_EPP1xxx.Beckhoff_EPP1xxxEK1122.A_0017_EPP1258_0002_0017.Latch.Status0 <-> Latch/Status0
//     PlcTask Inputs/GVL_iXlinker.EtherCAT_Master_EPPxxxx.Beckhoff_EPP1xxx.Beckhoff_EPP1xxxEK1122.A_0017_EPP1258_0002_0017.Latch.Status1 <-> Latch/Status1
//     PlcTask Inputs/GVL_iXlinker.EtherCAT_Master_EPPxxxx.Beckhoff_EPP1xxx.Beckhoff_EPP1xxxEK1122.A_0017_EPP1258_0002_0017.Latch.LatchPos0 <-> Latch/LatchPos0
//     PlcTask Inputs/GVL_iXlinker.EtherCAT_Master_EPPxxxx.Beckhoff_EPP1xxx.Beckhoff_EPP1xxxEK1122.A_0017_EPP1258_0002_0017.Latch.LatchPos1 <-> Latch/LatchPos1
//     PlcTask Inputs/GVL_iXlinker.EtherCAT_Master_EPPxxxx.Beckhoff_EPP1xxx.Beckhoff_EPP1xxxEK1122.A_0017_EPP1258_0002_0017.Latch.LatchNeg0 <-> Latch/LatchNeg0
//     PlcTask Inputs/GVL_iXlinker.EtherCAT_Master_EPPxxxx.Beckhoff_EPP1xxx.Beckhoff_EPP1xxxEK1122.A_0017_EPP1258_0002_0017.Latch.LatchNeg1 <-> Latch/LatchNeg1
//     PlcTask Inputs/GVL_iXlinker.EtherCAT_Master_EPPxxxx.Beckhoff_EPP1xxx.Beckhoff_EPP1xxxEK1122.A_0017_EPP1258_0002_0017.WcState.WcState0 <-> WcState/WcState0
//     PlcTask Inputs/GVL_iXlinker.EtherCAT_Master_EPPxxxx.Beckhoff_EPP1xxx.Beckhoff_EPP1xxxEK1122.A_0017_EPP1258_0002_0017.WcState.WcState1 <-> WcState/WcState1
//     PlcTask Inputs/GVL_iXlinker.EtherCAT_Master_EPPxxxx.Beckhoff_EPP1xxx.Beckhoff_EPP1xxxEK1122.A_0017_EPP1258_0002_0017.WcState.InputToggle0 <-> WcState/InputToggle0
//     PlcTask Inputs/GVL_iXlinker.EtherCAT_Master_EPPxxxx.Beckhoff_EPP1xxx.Beckhoff_EPP1xxxEK1122.A_0017_EPP1258_0002_0017.WcState.InputToggle1 <-> WcState/InputToggle1
//     PlcTask Inputs/GVL_iXlinker.EtherCAT_Master_EPPxxxx.Beckhoff_EPP1xxx.Beckhoff_EPP1xxxEK1122.A_0017_EPP1258_0002_0017.InfoData.DcOutputShift <-> InfoData/DcOutputShift
//     PlcTask Inputs/GVL_iXlinker.EtherCAT_Master_EPPxxxx.Beckhoff_EPP1xxx.Beckhoff_EPP1xxxEK1122.A_0017_EPP1258_0002_0017.InfoData.DcInputShift <-> InfoData/DcInputShift
//     PlcTask Inputs/GVL_iXlinker.EtherCAT_Master_EPPxxxx.Beckhoff_EPP1xxx.Beckhoff_EPP1xxxEK1122.A_0017_EPP1258_0002_0017.InfoData.State <-> InfoData/State
//   PLC/PLC Instance <-> EtherCAT Master EPPxxxx/Beckhoff EPP1xxx/Beckhoff EPP1xxxEK1122/A_0018(EPP1321-0060-0016)
//     PlcTask Inputs/GVL_iXlinker.EtherCAT_Master_EPPxxxx.Beckhoff_EPP1xxx.Beckhoff_EPP1xxxEK1122.A_0018_EPP1321_0060_0016.InfoData.State <-> InfoData/State
//   PLC/PLC Instance <-> EtherCAT Master EPPxxxx/Beckhoff EPP1xxx/Beckhoff EPP1xxxEK1122/A_0018(EPP1321-0060-0016)/A_0019(EPP1322-0001-0016)
//     PlcTask Inputs/GVL_iXlinker.EtherCAT_Master_EPPxxxx.Beckhoff_EPP1xxx.Beckhoff_EPP1xxxEK1122.A_0018_EPP1321_0060_0016.A_0019_EPP1322_0001_0016.InfoData.State <-> InfoData/State
//   PLC/PLC Instance <-> EtherCAT Master EPPxxxx/Beckhoff EPP1xxx/Beckhoff EPP1xxxEK1122/A_0018(EPP1321-0060-0016)/A_0019(EPP1322-0001-0016)/A_0020(EPP1322-0001-0017)
//     PlcTask Inputs/GVL_iXlinker.EtherCAT_Master_EPPxxxx.Beckhoff_EPP1xxx.Beckhoff_EPP1xxxEK1122.A_0018_EPP1321_0060_0016.A_0019_EPP1322_0001_0016.A_0020_EPP1322_0001_0017.InfoData.State <-> InfoData/State
//   PLC/PLC Instance <-> EtherCAT Master EPPxxxx/Beckhoff EPP1xxx/Beckhoff EPP1xxxEK1122/A_0018(EPP1321-0060-0016)/A_0019(EPP1322-0001-0016)/A_0020(EPP1322-0001-0017)/A_0021(EPP1332-0001-0016)
//     PlcTask Inputs/GVL_iXlinker.EtherCAT_Master_EPPxxxx.Beckhoff_EPP1xxx.Beckhoff_EPP1xxxEK1122.A_0018_EPP1321_0060_0016.A_0019_EPP1322_0001_0016.A_0020_EPP1322_0001_0017.A_0021_EPP1332_0001_0016.InfoData.State <-> InfoData/State
//   PLC/PLC Instance <-> EtherCAT Master EPPxxxx/Beckhoff EPP1xxx/Beckhoff EPP1xxxEK1122/A_0018(EPP1321-0060-0016)/A_0019(EPP1322-0001-0016)/A_0020(EPP1322-0001-0017)/A_0021(EPP1332-0001-0016)/A_0022(EPP1332-0001-0017)
//     PlcTask Inputs/GVL_iXlinker.EtherCAT_Master_EPPxxxx.Beckhoff_EPP1xxx.Beckhoff_EPP1xxxEK1122.A_0018_EPP1321_0060_0016.A_0019_EPP1322_0001_0016.A_0020_EPP1322_0001_0017.A_0021_EPP1332_0001_0016.A_0022_EPP1332_0001_0017.InfoData.State <-> InfoData/State
//   PLC/PLC Instance <-> EtherCAT Master EPPxxxx/Beckhoff EPP1xxx/Beckhoff EPP1xxxEK1122/A_0018(EPP1321-0060-0016)/A_0019(EPP1322-0001-0016)/A_0020(EPP1322-0001-0017)/A_0021(EPP1332-0001-0016)/A_0022(EPP1332-0001-0017)/A_0023(EPP1342-0001-0016)
//     PlcTask Inputs/GVL_iXlinker.EtherCAT_Master_EPPxxxx.Beckhoff_EPP1xxx.Beckhoff_EPP1xxxEK1122.A_0018_EPP1321_0060_0016.A_0019_EPP1322_0001_0016.A_0020_EPP1322_0001_0017.A_0021_EPP1332_0001_0016.A_0022_EPP1332_0001_0017.A_0023_EPP1342_0001_0016.InfoData.State <-> InfoData/State
//   PLC/PLC Instance <-> EtherCAT Master EPPxxxx/Beckhoff EPP1xxx/Beckhoff EPP1xxxEK1122/A_0018(EPP1321-0060-0016)/A_0019(EPP1322-0001-0016)/A_0020(EPP1322-0001-0017)/A_0021(EPP1332-0001-0016)/A_0022(EPP1332-0001-0017)/A_0023(EPP1342-0001-0016)/A_0024(EPP1342-0001-0017)
//     PlcTask Inputs/GVL_iXlinker.EtherCAT_Master_EPPxxxx.Beckhoff_EPP1xxx.Beckhoff_EPP1xxxEK1122.A_0018_EPP1321_0060_0016.A_0019_EPP1322_0001_0016.A_0020_EPP1322_0001_0017.A_0021_EPP1332_0001_0016.A_0022_EPP1332_0001_0017.A_0023_EPP1342_0001_0016.A_0024_EPP1342_0001_0017.InfoData.State <-> InfoData/State
//   PLC/PLC Instance <-> EtherCAT Master EPPxxxx/Beckhoff EPP1xxx/Beckhoff EPP1xxxEK1122/A_0018(EPP1321-0060-0016)/A_0019(EPP1322-0001-0016)/A_0020(EPP1322-0001-0017)/A_0021(EPP1332-0001-0016)/A_0022(EPP1332-0001-0017)/A_0023(EPP1342-0001-0016)/A_0024(EPP1342-0001-0017)/A_0025(EPP1518-0002-0016)
//     PlcTask Inputs/GVL_iXlinker.EtherCAT_Master_EPPxxxx.Beckhoff_EPP1xxx.Beckhoff_EPP1xxxEK1122.A_0018_EPP1321_0060_0016.A_0019_EPP1322_0001_0016.A_0020_EPP1322_0001_0017.A_0021_EPP1332_0001_0016.A_0022_EPP1332_0001_0017.A_0023_EPP1342_0001_0016.A_0024_EPP1342_0001_0017.A_0025_EPP1518_0002_0016.CNT_Input_Channel_1.Status/Set_counter_done <-> CNT Input Channel 1/Status/Set counter done
//     PlcTask Inputs/GVL_iXlinker.EtherCAT_Master_EPPxxxx.Beckhoff_EPP1xxx.Beckhoff_EPP1xxxEK1122.A_0018_EPP1321_0060_0016.A_0019_EPP1322_0001_0016.A_0020_EPP1322_0001_0017.A_0021_EPP1332_0001_0016.A_0022_EPP1332_0001_0017.A_0023_EPP1342_0001_0016.A_0024_EPP1342_0001_0017.A_0025_EPP1518_0002_0016.CNT_Input_Channel_2.Status/Set_counter_done <-> CNT Input Channel 2/Status/Set counter done
//     PlcTask Inputs/GVL_iXlinker.EtherCAT_Master_EPPxxxx.Beckhoff_EPP1xxx.Beckhoff_EPP1xxxEK1122.A_0018_EPP1321_0060_0016.A_0019_EPP1322_0001_0016.A_0020_EPP1322_0001_0017.A_0021_EPP1332_0001_0016.A_0022_EPP1332_0001_0017.A_0023_EPP1342_0001_0016.A_0024_EPP1342_0001_0017.A_0025_EPP1518_0002_0016.CNT_Input_Channel_1.Status/Counter_inhibited <-> CNT Input Channel 1/Status/Counter inhibited
//     PlcTask Inputs/GVL_iXlinker.EtherCAT_Master_EPPxxxx.Beckhoff_EPP1xxx.Beckhoff_EPP1xxxEK1122.A_0018_EPP1321_0060_0016.A_0019_EPP1322_0001_0016.A_0020_EPP1322_0001_0017.A_0021_EPP1332_0001_0016.A_0022_EPP1332_0001_0017.A_0023_EPP1342_0001_0016.A_0024_EPP1342_0001_0017.A_0025_EPP1518_0002_0016.CNT_Input_Channel_2.Status/Counter_inhibited <-> CNT Input Channel 2/Status/Counter inhibited
//     PlcTask Inputs/GVL_iXlinker.EtherCAT_Master_EPPxxxx.Beckhoff_EPP1xxx.Beckhoff_EPP1xxxEK1122.A_0018_EPP1321_0060_0016.A_0019_EPP1322_0001_0016.A_0020_EPP1322_0001_0017.A_0021_EPP1332_0001_0016.A_0022_EPP1332_0001_0017.A_0023_EPP1342_0001_0016.A_0024_EPP1342_0001_0017.A_0025_EPP1518_0002_0016.CNT_Input_Channel_1.Status/Status_of_input_UD <-> CNT Input Channel 1/Status/Status of input UD
//     PlcTask Inputs/GVL_iXlinker.EtherCAT_Master_EPPxxxx.Beckhoff_EPP1xxx.Beckhoff_EPP1xxxEK1122.A_0018_EPP1321_0060_0016.A_0019_EPP1322_0001_0016.A_0020_EPP1322_0001_0017.A_0021_EPP1332_0001_0016.A_0022_EPP1332_0001_0017.A_0023_EPP1342_0001_0016.A_0024_EPP1342_0001_0017.A_0025_EPP1518_0002_0016.CNT_Input_Channel_2.Status/Status_of_input_UD <-> CNT Input Channel 2/Status/Status of input UD
//     PlcTask Inputs/GVL_iXlinker.EtherCAT_Master_EPPxxxx.Beckhoff_EPP1xxx.Beckhoff_EPP1xxxEK1122.A_0018_EPP1321_0060_0016.A_0019_EPP1322_0001_0016.A_0020_EPP1322_0001_0017.A_0021_EPP1332_0001_0016.A_0022_EPP1332_0001_0017.A_0023_EPP1342_0001_0016.A_0024_EPP1342_0001_0017.A_0025_EPP1518_0002_0016.CNT_Input_Channel_1.Status/Status_of_input_clock <-> CNT Input Channel 1/Status/Status of input clock
//     PlcTask Inputs/GVL_iXlinker.EtherCAT_Master_EPPxxxx.Beckhoff_EPP1xxx.Beckhoff_EPP1xxxEK1122.A_0018_EPP1321_0060_0016.A_0019_EPP1322_0001_0016.A_0020_EPP1322_0001_0017.A_0021_EPP1332_0001_0016.A_0022_EPP1332_0001_0017.A_0023_EPP1342_0001_0016.A_0024_EPP1342_0001_0017.A_0025_EPP1518_0002_0016.CNT_Input_Channel_2.Status/Status_of_input_clock <-> CNT Input Channel 2/Status/Status of input clock
//     PlcTask Inputs/GVL_iXlinker.EtherCAT_Master_EPPxxxx.Beckhoff_EPP1xxx.Beckhoff_EPP1xxxEK1122.A_0018_EPP1321_0060_0016.A_0019_EPP1322_0001_0016.A_0020_EPP1322_0001_0017.A_0021_EPP1332_0001_0016.A_0022_EPP1332_0001_0017.A_0023_EPP1342_0001_0016.A_0024_EPP1342_0001_0017.A_0025_EPP1518_0002_0016.CNT_Input_Channel_1.Status/Sync_error <-> CNT Input Channel 1/Status/Sync error
//     PlcTask Inputs/GVL_iXlinker.EtherCAT_Master_EPPxxxx.Beckhoff_EPP1xxx.Beckhoff_EPP1xxxEK1122.A_0018_EPP1321_0060_0016.A_0019_EPP1322_0001_0016.A_0020_EPP1322_0001_0017.A_0021_EPP1332_0001_0016.A_0022_EPP1332_0001_0017.A_0023_EPP1342_0001_0016.A_0024_EPP1342_0001_0017.A_0025_EPP1518_0002_0016.CNT_Input_Channel_2.Status/Sync_error <-> CNT Input Channel 2/Status/Sync error
//     PlcTask Inputs/GVL_iXlinker.EtherCAT_Master_EPPxxxx.Beckhoff_EPP1xxx.Beckhoff_EPP1xxxEK1122.A_0018_EPP1321_0060_0016.A_0019_EPP1322_0001_0016.A_0020_EPP1322_0001_0017.A_0021_EPP1332_0001_0016.A_0022_EPP1332_0001_0017.A_0023_EPP1342_0001_0016.A_0024_EPP1342_0001_0017.A_0025_EPP1518_0002_0016.CNT_Input_Channel_1.Status/TxPDO_State <-> CNT Input Channel 1/Status/TxPDO State
//     PlcTask Inputs/GVL_iXlinker.EtherCAT_Master_EPPxxxx.Beckhoff_EPP1xxx.Beckhoff_EPP1xxxEK1122.A_0018_EPP1321_0060_0016.A_0019_EPP1322_0001_0016.A_0020_EPP1322_0001_0017.A_0021_EPP1332_0001_0016.A_0022_EPP1332_0001_0017.A_0023_EPP1342_0001_0016.A_0024_EPP1342_0001_0017.A_0025_EPP1518_0002_0016.CNT_Input_Channel_2.Status/TxPDO_State <-> CNT Input Channel 2/Status/TxPDO State
//     PlcTask Inputs/GVL_iXlinker.EtherCAT_Master_EPPxxxx.Beckhoff_EPP1xxx.Beckhoff_EPP1xxxEK1122.A_0018_EPP1321_0060_0016.A_0019_EPP1322_0001_0016.A_0020_EPP1322_0001_0017.A_0021_EPP1332_0001_0016.A_0022_EPP1332_0001_0017.A_0023_EPP1342_0001_0016.A_0024_EPP1342_0001_0017.A_0025_EPP1518_0002_0016.CNT_Input_Channel_1.Status/TxPDO_Toggle <-> CNT Input Channel 1/Status/TxPDO Toggle
//     PlcTask Inputs/GVL_iXlinker.EtherCAT_Master_EPPxxxx.Beckhoff_EPP1xxx.Beckhoff_EPP1xxxEK1122.A_0018_EPP1321_0060_0016.A_0019_EPP1322_0001_0016.A_0020_EPP1322_0001_0017.A_0021_EPP1332_0001_0016.A_0022_EPP1332_0001_0017.A_0023_EPP1342_0001_0016.A_0024_EPP1342_0001_0017.A_0025_EPP1518_0002_0016.CNT_Input_Channel_2.Status/TxPDO_Toggle <-> CNT Input Channel 2/Status/TxPDO Toggle
//     PlcTask Inputs/GVL_iXlinker.EtherCAT_Master_EPPxxxx.Beckhoff_EPP1xxx.Beckhoff_EPP1xxxEK1122.A_0018_EPP1321_0060_0016.A_0019_EPP1322_0001_0016.A_0020_EPP1322_0001_0017.A_0021_EPP1332_0001_0016.A_0022_EPP1332_0001_0017.A_0023_EPP1342_0001_0016.A_0024_EPP1342_0001_0017.A_0025_EPP1518_0002_0016.CNT_Input_Channel_1.Counter_value <-> CNT Input Channel 1/Counter value
//     PlcTask Inputs/GVL_iXlinker.EtherCAT_Master_EPPxxxx.Beckhoff_EPP1xxx.Beckhoff_EPP1xxxEK1122.A_0018_EPP1321_0060_0016.A_0019_EPP1322_0001_0016.A_0020_EPP1322_0001_0017.A_0021_EPP1332_0001_0016.A_0022_EPP1332_0001_0017.A_0023_EPP1342_0001_0016.A_0024_EPP1342_0001_0017.A_0025_EPP1518_0002_0016.CNT_Input_Channel_2.Counter_value <-> CNT Input Channel 2/Counter value
//     PlcTask Inputs/GVL_iXlinker.EtherCAT_Master_EPPxxxx.Beckhoff_EPP1xxx.Beckhoff_EPP1xxxEK1122.A_0018_EPP1321_0060_0016.A_0019_EPP1322_0001_0016.A_0020_EPP1322_0001_0017.A_0021_EPP1332_0001_0016.A_0022_EPP1332_0001_0017.A_0023_EPP1342_0001_0016.A_0024_EPP1342_0001_0017.A_0025_EPP1518_0002_0016.DIG_Inputs.Input[0] <-> DIG Inputs/Input 0
//     PlcTask Inputs/GVL_iXlinker.EtherCAT_Master_EPPxxxx.Beckhoff_EPP1xxx.Beckhoff_EPP1xxxEK1122.A_0018_EPP1321_0060_0016.A_0019_EPP1322_0001_0016.A_0020_EPP1322_0001_0017.A_0021_EPP1332_0001_0016.A_0022_EPP1332_0001_0017.A_0023_EPP1342_0001_0016.A_0024_EPP1342_0001_0017.A_0025_EPP1518_0002_0016.DIG_Inputs.Input[1] <-> DIG Inputs/Input 1
//     PlcTask Inputs/GVL_iXlinker.EtherCAT_Master_EPPxxxx.Beckhoff_EPP1xxx.Beckhoff_EPP1xxxEK1122.A_0018_EPP1321_0060_0016.A_0019_EPP1322_0001_0016.A_0020_EPP1322_0001_0017.A_0021_EPP1332_0001_0016.A_0022_EPP1332_0001_0017.A_0023_EPP1342_0001_0016.A_0024_EPP1342_0001_0017.A_0025_EPP1518_0002_0016.DIG_Inputs.Input[2] <-> DIG Inputs/Input 2
//     PlcTask Inputs/GVL_iXlinker.EtherCAT_Master_EPPxxxx.Beckhoff_EPP1xxx.Beckhoff_EPP1xxxEK1122.A_0018_EPP1321_0060_0016.A_0019_EPP1322_0001_0016.A_0020_EPP1322_0001_0017.A_0021_EPP1332_0001_0016.A_0022_EPP1332_0001_0017.A_0023_EPP1342_0001_0016.A_0024_EPP1342_0001_0017.A_0025_EPP1518_0002_0016.DIG_Inputs.Input[3] <-> DIG Inputs/Input 3
//     PlcTask Inputs/GVL_iXlinker.EtherCAT_Master_EPPxxxx.Beckhoff_EPP1xxx.Beckhoff_EPP1xxxEK1122.A_0018_EPP1321_0060_0016.A_0019_EPP1322_0001_0016.A_0020_EPP1322_0001_0017.A_0021_EPP1332_0001_0016.A_0022_EPP1332_0001_0017.A_0023_EPP1342_0001_0016.A_0024_EPP1342_0001_0017.A_0025_EPP1518_0002_0016.DIG_Inputs.Input[4] <-> DIG Inputs/Input 4
//     PlcTask Inputs/GVL_iXlinker.EtherCAT_Master_EPPxxxx.Beckhoff_EPP1xxx.Beckhoff_EPP1xxxEK1122.A_0018_EPP1321_0060_0016.A_0019_EPP1322_0001_0016.A_0020_EPP1322_0001_0017.A_0021_EPP1332_0001_0016.A_0022_EPP1332_0001_0017.A_0023_EPP1342_0001_0016.A_0024_EPP1342_0001_0017.A_0025_EPP1518_0002_0016.DIG_Inputs.Input[5] <-> DIG Inputs/Input 5
//     PlcTask Inputs/GVL_iXlinker.EtherCAT_Master_EPPxxxx.Beckhoff_EPP1xxx.Beckhoff_EPP1xxxEK1122.A_0018_EPP1321_0060_0016.A_0019_EPP1322_0001_0016.A_0020_EPP1322_0001_0017.A_0021_EPP1332_0001_0016.A_0022_EPP1332_0001_0017.A_0023_EPP1342_0001_0016.A_0024_EPP1342_0001_0017.A_0025_EPP1518_0002_0016.DIG_Inputs.Input[6] <-> DIG Inputs/Input 6
//     PlcTask Inputs/GVL_iXlinker.EtherCAT_Master_EPPxxxx.Beckhoff_EPP1xxx.Beckhoff_EPP1xxxEK1122.A_0018_EPP1321_0060_0016.A_0019_EPP1322_0001_0016.A_0020_EPP1322_0001_0017.A_0021_EPP1332_0001_0016.A_0022_EPP1332_0001_0017.A_0023_EPP1342_0001_0016.A_0024_EPP1342_0001_0017.A_0025_EPP1518_0002_0016.DIG_Inputs.Input[7] <-> DIG Inputs/Input 7
//     PlcTask Inputs/GVL_iXlinker.EtherCAT_Master_EPPxxxx.Beckhoff_EPP1xxx.Beckhoff_EPP1xxxEK1122.A_0018_EPP1321_0060_0016.A_0019_EPP1322_0001_0016.A_0020_EPP1322_0001_0017.A_0021_EPP1332_0001_0016.A_0022_EPP1332_0001_0017.A_0023_EPP1342_0001_0016.A_0024_EPP1342_0001_0017.A_0025_EPP1518_0002_0016.DIG_Inputs_Device.Status/Error_channel_1 <-> DIG Inputs Device/Status/Error channel 1
//     PlcTask Inputs/GVL_iXlinker.EtherCAT_Master_EPPxxxx.Beckhoff_EPP1xxx.Beckhoff_EPP1xxxEK1122.A_0018_EPP1321_0060_0016.A_0019_EPP1322_0001_0016.A_0020_EPP1322_0001_0017.A_0021_EPP1332_0001_0016.A_0022_EPP1332_0001_0017.A_0023_EPP1342_0001_0016.A_0024_EPP1342_0001_0017.A_0025_EPP1518_0002_0016.DIG_Inputs_Device.Status/Error_channel_2 <-> DIG Inputs Device/Status/Error channel 2
//     PlcTask Inputs/GVL_iXlinker.EtherCAT_Master_EPPxxxx.Beckhoff_EPP1xxx.Beckhoff_EPP1xxxEK1122.A_0018_EPP1321_0060_0016.A_0019_EPP1322_0001_0016.A_0020_EPP1322_0001_0017.A_0021_EPP1332_0001_0016.A_0022_EPP1332_0001_0017.A_0023_EPP1342_0001_0016.A_0024_EPP1342_0001_0017.A_0025_EPP1518_0002_0016.DIG_Inputs_Device.Status/Sync_error <-> DIG Inputs Device/Status/Sync error
//     PlcTask Inputs/GVL_iXlinker.EtherCAT_Master_EPPxxxx.Beckhoff_EPP1xxx.Beckhoff_EPP1xxxEK1122.A_0018_EPP1321_0060_0016.A_0019_EPP1322_0001_0016.A_0020_EPP1322_0001_0017.A_0021_EPP1332_0001_0016.A_0022_EPP1332_0001_0017.A_0023_EPP1342_0001_0016.A_0024_EPP1342_0001_0017.A_0025_EPP1518_0002_0016.DIG_Inputs_Device.Status/TxPDO_State <-> DIG Inputs Device/Status/TxPDO State
//     PlcTask Inputs/GVL_iXlinker.EtherCAT_Master_EPPxxxx.Beckhoff_EPP1xxx.Beckhoff_EPP1xxxEK1122.A_0018_EPP1321_0060_0016.A_0019_EPP1322_0001_0016.A_0020_EPP1322_0001_0017.A_0021_EPP1332_0001_0016.A_0022_EPP1332_0001_0017.A_0023_EPP1342_0001_0016.A_0024_EPP1342_0001_0017.A_0025_EPP1518_0002_0016.DIG_Inputs_Device.Status/TxPDO_Toggle <-> DIG Inputs Device/Status/TxPDO Toggle
//     PlcTask Outputs/GVL_iXlinker.EtherCAT_Master_EPPxxxx.Beckhoff_EPP1xxx.Beckhoff_EPP1xxxEK1122.A_0018_EPP1321_0060_0016.A_0019_EPP1322_0001_0016.A_0020_EPP1322_0001_0017.A_0021_EPP1332_0001_0016.A_0022_EPP1332_0001_0017.A_0023_EPP1342_0001_0016.A_0024_EPP1342_0001_0017.A_0025_EPP1518_0002_0016.CNT_Output_Channel_1.Control/Set_counter <-> CNT Output Channel 1/Control/Set counter
//     PlcTask Outputs/GVL_iXlinker.EtherCAT_Master_EPPxxxx.Beckhoff_EPP1xxx.Beckhoff_EPP1xxxEK1122.A_0018_EPP1321_0060_0016.A_0019_EPP1322_0001_0016.A_0020_EPP1322_0001_0017.A_0021_EPP1332_0001_0016.A_0022_EPP1332_0001_0017.A_0023_EPP1342_0001_0016.A_0024_EPP1342_0001_0017.A_0025_EPP1518_0002_0016.CNT_Output_Channel_2.Control/Set_counter <-> CNT Output Channel 2/Control/Set counter
//     PlcTask Outputs/GVL_iXlinker.EtherCAT_Master_EPPxxxx.Beckhoff_EPP1xxx.Beckhoff_EPP1xxxEK1122.A_0018_EPP1321_0060_0016.A_0019_EPP1322_0001_0016.A_0020_EPP1322_0001_0017.A_0021_EPP1332_0001_0016.A_0022_EPP1332_0001_0017.A_0023_EPP1342_0001_0016.A_0024_EPP1342_0001_0017.A_0025_EPP1518_0002_0016.CNT_Output_Channel_1.Control/Inhibit_counter <-> CNT Output Channel 1/Control/Inhibit counter
//     PlcTask Outputs/GVL_iXlinker.EtherCAT_Master_EPPxxxx.Beckhoff_EPP1xxx.Beckhoff_EPP1xxxEK1122.A_0018_EPP1321_0060_0016.A_0019_EPP1322_0001_0016.A_0020_EPP1322_0001_0017.A_0021_EPP1332_0001_0016.A_0022_EPP1332_0001_0017.A_0023_EPP1342_0001_0016.A_0024_EPP1342_0001_0017.A_0025_EPP1518_0002_0016.CNT_Output_Channel_2.Control/Inhibit_counter <-> CNT Output Channel 2/Control/Inhibit counter
//     PlcTask Outputs/GVL_iXlinker.EtherCAT_Master_EPPxxxx.Beckhoff_EPP1xxx.Beckhoff_EPP1xxxEK1122.A_0018_EPP1321_0060_0016.A_0019_EPP1322_0001_0016.A_0020_EPP1322_0001_0017.A_0021_EPP1332_0001_0016.A_0022_EPP1332_0001_0017.A_0023_EPP1342_0001_0016.A_0024_EPP1342_0001_0017.A_0025_EPP1518_0002_0016.CNT_Output_Channel_1.Set_counter_value <-> CNT Output Channel 1/Set counter value
//     PlcTask Outputs/GVL_iXlinker.EtherCAT_Master_EPPxxxx.Beckhoff_EPP1xxx.Beckhoff_EPP1xxxEK1122.A_0018_EPP1321_0060_0016.A_0019_EPP1322_0001_0016.A_0020_EPP1322_0001_0017.A_0021_EPP1332_0001_0016.A_0022_EPP1332_0001_0017.A_0023_EPP1342_0001_0016.A_0024_EPP1342_0001_0017.A_0025_EPP1518_0002_0016.CNT_Output_Channel_2.Set_counter_value <-> CNT Output Channel 2/Set counter value
//     PlcTask Inputs/GVL_iXlinker.EtherCAT_Master_EPPxxxx.Beckhoff_EPP1xxx.Beckhoff_EPP1xxxEK1122.A_0018_EPP1321_0060_0016.A_0019_EPP1322_0001_0016.A_0020_EPP1322_0001_0017.A_0021_EPP1332_0001_0016.A_0022_EPP1332_0001_0017.A_0023_EPP1342_0001_0016.A_0024_EPP1342_0001_0017.A_0025_EPP1518_0002_0016.WcState.WcState <-> WcState/WcState
//     PlcTask Inputs/GVL_iXlinker.EtherCAT_Master_EPPxxxx.Beckhoff_EPP1xxx.Beckhoff_EPP1xxxEK1122.A_0018_EPP1321_0060_0016.A_0019_EPP1322_0001_0016.A_0020_EPP1322_0001_0017.A_0021_EPP1332_0001_0016.A_0022_EPP1332_0001_0017.A_0023_EPP1342_0001_0016.A_0024_EPP1342_0001_0017.A_0025_EPP1518_0002_0016.WcState.InputToggle <-> WcState/InputToggle
//     PlcTask Inputs/GVL_iXlinker.EtherCAT_Master_EPPxxxx.Beckhoff_EPP1xxx.Beckhoff_EPP1xxxEK1122.A_0018_EPP1321_0060_0016.A_0019_EPP1322_0001_0016.A_0020_EPP1322_0001_0017.A_0021_EPP1332_0001_0016.A_0022_EPP1332_0001_0017.A_0023_EPP1342_0001_0016.A_0024_EPP1342_0001_0017.A_0025_EPP1518_0002_0016.InfoData.AdsAddr <-> InfoData/AdsAddr
//     PlcTask Inputs/GVL_iXlinker.EtherCAT_Master_EPPxxxx.Beckhoff_EPP1xxx.Beckhoff_EPP1xxxEK1122.A_0018_EPP1321_0060_0016.A_0019_EPP1322_0001_0016.A_0020_EPP1322_0001_0017.A_0021_EPP1332_0001_0016.A_0022_EPP1332_0001_0017.A_0023_EPP1342_0001_0016.A_0024_EPP1342_0001_0017.A_0025_EPP1518_0002_0016.InfoData.State <-> InfoData/State
//   PLC/PLC Instance <-> EtherCAT Master EPPxxxx/Beckhoff EPP1xxx/Beckhoff EPP1xxxEK1122/A_0018(EPP1321-0060-0016)/A_0019(EPP1322-0001-0016)/A_0020(EPP1322-0001-0017)/A_0021(EPP1332-0001-0016)/A_0022(EPP1332-0001-0017)/A_0023(EPP1342-0001-0016)/A_0024(EPP1342-0001-0017)/A_0026(EPP1518-0002-0017)
//     PlcTask Inputs/GVL_iXlinker.EtherCAT_Master_EPPxxxx.Beckhoff_EPP1xxx.Beckhoff_EPP1xxxEK1122.A_0018_EPP1321_0060_0016.A_0019_EPP1322_0001_0016.A_0020_EPP1322_0001_0017.A_0021_EPP1332_0001_0016.A_0022_EPP1332_0001_0017.A_0023_EPP1342_0001_0016.A_0024_EPP1342_0001_0017.A_0026_EPP1518_0002_0017.CNT_Input_Channel_1.Status/Set_counter_done <-> CNT Input Channel 1/Status/Set counter done
//     PlcTask Inputs/GVL_iXlinker.EtherCAT_Master_EPPxxxx.Beckhoff_EPP1xxx.Beckhoff_EPP1xxxEK1122.A_0018_EPP1321_0060_0016.A_0019_EPP1322_0001_0016.A_0020_EPP1322_0001_0017.A_0021_EPP1332_0001_0016.A_0022_EPP1332_0001_0017.A_0023_EPP1342_0001_0016.A_0024_EPP1342_0001_0017.A_0026_EPP1518_0002_0017.CNT_Input_Channel_2.Status/Set_counter_done <-> CNT Input Channel 2/Status/Set counter done
//     PlcTask Inputs/GVL_iXlinker.EtherCAT_Master_EPPxxxx.Beckhoff_EPP1xxx.Beckhoff_EPP1xxxEK1122.A_0018_EPP1321_0060_0016.A_0019_EPP1322_0001_0016.A_0020_EPP1322_0001_0017.A_0021_EPP1332_0001_0016.A_0022_EPP1332_0001_0017.A_0023_EPP1342_0001_0016.A_0024_EPP1342_0001_0017.A_0026_EPP1518_0002_0017.CNT_Input_Channel_1.Status/Counter_inhibited <-> CNT Input Channel 1/Status/Counter inhibited
//     PlcTask Inputs/GVL_iXlinker.EtherCAT_Master_EPPxxxx.Beckhoff_EPP1xxx.Beckhoff_EPP1xxxEK1122.A_0018_EPP1321_0060_0016.A_0019_EPP1322_0001_0016.A_0020_EPP1322_0001_0017.A_0021_EPP1332_0001_0016.A_0022_EPP1332_0001_0017.A_0023_EPP1342_0001_0016.A_0024_EPP1342_0001_0017.A_0026_EPP1518_0002_0017.CNT_Input_Channel_2.Status/Counter_inhibited <-> CNT Input Channel 2/Status/Counter inhibited
//     PlcTask Inputs/GVL_iXlinker.EtherCAT_Master_EPPxxxx.Beckhoff_EPP1xxx.Beckhoff_EPP1xxxEK1122.A_0018_EPP1321_0060_0016.A_0019_EPP1322_0001_0016.A_0020_EPP1322_0001_0017.A_0021_EPP1332_0001_0016.A_0022_EPP1332_0001_0017.A_0023_EPP1342_0001_0016.A_0024_EPP1342_0001_0017.A_0026_EPP1518_0002_0017.CNT_Input_Channel_1.Status/Status_of_input_UD <-> CNT Input Channel 1/Status/Status of input UD
//     PlcTask Inputs/GVL_iXlinker.EtherCAT_Master_EPPxxxx.Beckhoff_EPP1xxx.Beckhoff_EPP1xxxEK1122.A_0018_EPP1321_0060_0016.A_0019_EPP1322_0001_0016.A_0020_EPP1322_0001_0017.A_0021_EPP1332_0001_0016.A_0022_EPP1332_0001_0017.A_0023_EPP1342_0001_0016.A_0024_EPP1342_0001_0017.A_0026_EPP1518_0002_0017.CNT_Input_Channel_2.Status/Status_of_input_UD <-> CNT Input Channel 2/Status/Status of input UD
//     PlcTask Inputs/GVL_iXlinker.EtherCAT_Master_EPPxxxx.Beckhoff_EPP1xxx.Beckhoff_EPP1xxxEK1122.A_0018_EPP1321_0060_0016.A_0019_EPP1322_0001_0016.A_0020_EPP1322_0001_0017.A_0021_EPP1332_0001_0016.A_0022_EPP1332_0001_0017.A_0023_EPP1342_0001_0016.A_0024_EPP1342_0001_0017.A_0026_EPP1518_0002_0017.CNT_Input_Channel_1.Status/Status_of_input_clock <-> CNT Input Channel 1/Status/Status of input clock
//     PlcTask Inputs/GVL_iXlinker.EtherCAT_Master_EPPxxxx.Beckhoff_EPP1xxx.Beckhoff_EPP1xxxEK1122.A_0018_EPP1321_0060_0016.A_0019_EPP1322_0001_0016.A_0020_EPP1322_0001_0017.A_0021_EPP1332_0001_0016.A_0022_EPP1332_0001_0017.A_0023_EPP1342_0001_0016.A_0024_EPP1342_0001_0017.A_0026_EPP1518_0002_0017.CNT_Input_Channel_2.Status/Status_of_input_clock <-> CNT Input Channel 2/Status/Status of input clock
//     PlcTask Inputs/GVL_iXlinker.EtherCAT_Master_EPPxxxx.Beckhoff_EPP1xxx.Beckhoff_EPP1xxxEK1122.A_0018_EPP1321_0060_0016.A_0019_EPP1322_0001_0016.A_0020_EPP1322_0001_0017.A_0021_EPP1332_0001_0016.A_0022_EPP1332_0001_0017.A_0023_EPP1342_0001_0016.A_0024_EPP1342_0001_0017.A_0026_EPP1518_0002_0017.CNT_Input_Channel_1.Status/Sync_error <-> CNT Input Channel 1/Status/Sync error
//     PlcTask Inputs/GVL_iXlinker.EtherCAT_Master_EPPxxxx.Beckhoff_EPP1xxx.Beckhoff_EPP1xxxEK1122.A_0018_EPP1321_0060_0016.A_0019_EPP1322_0001_0016.A_0020_EPP1322_0001_0017.A_0021_EPP1332_0001_0016.A_0022_EPP1332_0001_0017.A_0023_EPP1342_0001_0016.A_0024_EPP1342_0001_0017.A_0026_EPP1518_0002_0017.CNT_Input_Channel_2.Status/Sync_error <-> CNT Input Channel 2/Status/Sync error
//     PlcTask Inputs/GVL_iXlinker.EtherCAT_Master_EPPxxxx.Beckhoff_EPP1xxx.Beckhoff_EPP1xxxEK1122.A_0018_EPP1321_0060_0016.A_0019_EPP1322_0001_0016.A_0020_EPP1322_0001_0017.A_0021_EPP1332_0001_0016.A_0022_EPP1332_0001_0017.A_0023_EPP1342_0001_0016.A_0024_EPP1342_0001_0017.A_0026_EPP1518_0002_0017.CNT_Input_Channel_1.Status/TxPDO_State <-> CNT Input Channel 1/Status/TxPDO State
//     PlcTask Inputs/GVL_iXlinker.EtherCAT_Master_EPPxxxx.Beckhoff_EPP1xxx.Beckhoff_EPP1xxxEK1122.A_0018_EPP1321_0060_0016.A_0019_EPP1322_0001_0016.A_0020_EPP1322_0001_0017.A_0021_EPP1332_0001_0016.A_0022_EPP1332_0001_0017.A_0023_EPP1342_0001_0016.A_0024_EPP1342_0001_0017.A_0026_EPP1518_0002_0017.CNT_Input_Channel_2.Status/TxPDO_State <-> CNT Input Channel 2/Status/TxPDO State
//     PlcTask Inputs/GVL_iXlinker.EtherCAT_Master_EPPxxxx.Beckhoff_EPP1xxx.Beckhoff_EPP1xxxEK1122.A_0018_EPP1321_0060_0016.A_0019_EPP1322_0001_0016.A_0020_EPP1322_0001_0017.A_0021_EPP1332_0001_0016.A_0022_EPP1332_0001_0017.A_0023_EPP1342_0001_0016.A_0024_EPP1342_0001_0017.A_0026_EPP1518_0002_0017.CNT_Input_Channel_1.Status/TxPDO_Toggle <-> CNT Input Channel 1/Status/TxPDO Toggle
//     PlcTask Inputs/GVL_iXlinker.EtherCAT_Master_EPPxxxx.Beckhoff_EPP1xxx.Beckhoff_EPP1xxxEK1122.A_0018_EPP1321_0060_0016.A_0019_EPP1322_0001_0016.A_0020_EPP1322_0001_0017.A_0021_EPP1332_0001_0016.A_0022_EPP1332_0001_0017.A_0023_EPP1342_0001_0016.A_0024_EPP1342_0001_0017.A_0026_EPP1518_0002_0017.CNT_Input_Channel_2.Status/TxPDO_Toggle <-> CNT Input Channel 2/Status/TxPDO Toggle
//     PlcTask Inputs/GVL_iXlinker.EtherCAT_Master_EPPxxxx.Beckhoff_EPP1xxx.Beckhoff_EPP1xxxEK1122.A_0018_EPP1321_0060_0016.A_0019_EPP1322_0001_0016.A_0020_EPP1322_0001_0017.A_0021_EPP1332_0001_0016.A_0022_EPP1332_0001_0017.A_0023_EPP1342_0001_0016.A_0024_EPP1342_0001_0017.A_0026_EPP1518_0002_0017.CNT_Input_Channel_1.Counter_value <-> CNT Input Channel 1/Counter value
//     PlcTask Inputs/GVL_iXlinker.EtherCAT_Master_EPPxxxx.Beckhoff_EPP1xxx.Beckhoff_EPP1xxxEK1122.A_0018_EPP1321_0060_0016.A_0019_EPP1322_0001_0016.A_0020_EPP1322_0001_0017.A_0021_EPP1332_0001_0016.A_0022_EPP1332_0001_0017.A_0023_EPP1342_0001_0016.A_0024_EPP1342_0001_0017.A_0026_EPP1518_0002_0017.CNT_Input_Channel_2.Counter_value <-> CNT Input Channel 2/Counter value
//     PlcTask Inputs/GVL_iXlinker.EtherCAT_Master_EPPxxxx.Beckhoff_EPP1xxx.Beckhoff_EPP1xxxEK1122.A_0018_EPP1321_0060_0016.A_0019_EPP1322_0001_0016.A_0020_EPP1322_0001_0017.A_0021_EPP1332_0001_0016.A_0022_EPP1332_0001_0017.A_0023_EPP1342_0001_0016.A_0024_EPP1342_0001_0017.A_0026_EPP1518_0002_0017.DIG_Inputs.Input[0] <-> DIG Inputs/Input 0
//     PlcTask Inputs/GVL_iXlinker.EtherCAT_Master_EPPxxxx.Beckhoff_EPP1xxx.Beckhoff_EPP1xxxEK1122.A_0018_EPP1321_0060_0016.A_0019_EPP1322_0001_0016.A_0020_EPP1322_0001_0017.A_0021_EPP1332_0001_0016.A_0022_EPP1332_0001_0017.A_0023_EPP1342_0001_0016.A_0024_EPP1342_0001_0017.A_0026_EPP1518_0002_0017.DIG_Inputs.Input[1] <-> DIG Inputs/Input 1
//     PlcTask Inputs/GVL_iXlinker.EtherCAT_Master_EPPxxxx.Beckhoff_EPP1xxx.Beckhoff_EPP1xxxEK1122.A_0018_EPP1321_0060_0016.A_0019_EPP1322_0001_0016.A_0020_EPP1322_0001_0017.A_0021_EPP1332_0001_0016.A_0022_EPP1332_0001_0017.A_0023_EPP1342_0001_0016.A_0024_EPP1342_0001_0017.A_0026_EPP1518_0002_0017.DIG_Inputs.Input[2] <-> DIG Inputs/Input 2
//     PlcTask Inputs/GVL_iXlinker.EtherCAT_Master_EPPxxxx.Beckhoff_EPP1xxx.Beckhoff_EPP1xxxEK1122.A_0018_EPP1321_0060_0016.A_0019_EPP1322_0001_0016.A_0020_EPP1322_0001_0017.A_0021_EPP1332_0001_0016.A_0022_EPP1332_0001_0017.A_0023_EPP1342_0001_0016.A_0024_EPP1342_0001_0017.A_0026_EPP1518_0002_0017.DIG_Inputs.Input[3] <-> DIG Inputs/Input 3
//     PlcTask Inputs/GVL_iXlinker.EtherCAT_Master_EPPxxxx.Beckhoff_EPP1xxx.Beckhoff_EPP1xxxEK1122.A_0018_EPP1321_0060_0016.A_0019_EPP1322_0001_0016.A_0020_EPP1322_0001_0017.A_0021_EPP1332_0001_0016.A_0022_EPP1332_0001_0017.A_0023_EPP1342_0001_0016.A_0024_EPP1342_0001_0017.A_0026_EPP1518_0002_0017.DIG_Inputs.Input[4] <-> DIG Inputs/Input 4
//     PlcTask Inputs/GVL_iXlinker.EtherCAT_Master_EPPxxxx.Beckhoff_EPP1xxx.Beckhoff_EPP1xxxEK1122.A_0018_EPP1321_0060_0016.A_0019_EPP1322_0001_0016.A_0020_EPP1322_0001_0017.A_0021_EPP1332_0001_0016.A_0022_EPP1332_0001_0017.A_0023_EPP1342_0001_0016.A_0024_EPP1342_0001_0017.A_0026_EPP1518_0002_0017.DIG_Inputs.Input[5] <-> DIG Inputs/Input 5
//     PlcTask Inputs/GVL_iXlinker.EtherCAT_Master_EPPxxxx.Beckhoff_EPP1xxx.Beckhoff_EPP1xxxEK1122.A_0018_EPP1321_0060_0016.A_0019_EPP1322_0001_0016.A_0020_EPP1322_0001_0017.A_0021_EPP1332_0001_0016.A_0022_EPP1332_0001_0017.A_0023_EPP1342_0001_0016.A_0024_EPP1342_0001_0017.A_0026_EPP1518_0002_0017.DIG_Inputs.Input[6] <-> DIG Inputs/Input 6
//     PlcTask Inputs/GVL_iXlinker.EtherCAT_Master_EPPxxxx.Beckhoff_EPP1xxx.Beckhoff_EPP1xxxEK1122.A_0018_EPP1321_0060_0016.A_0019_EPP1322_0001_0016.A_0020_EPP1322_0001_0017.A_0021_EPP1332_0001_0016.A_0022_EPP1332_0001_0017.A_0023_EPP1342_0001_0016.A_0024_EPP1342_0001_0017.A_0026_EPP1518_0002_0017.DIG_Inputs.Input[7] <-> DIG Inputs/Input 7
//     PlcTask Inputs/GVL_iXlinker.EtherCAT_Master_EPPxxxx.Beckhoff_EPP1xxx.Beckhoff_EPP1xxxEK1122.A_0018_EPP1321_0060_0016.A_0019_EPP1322_0001_0016.A_0020_EPP1322_0001_0017.A_0021_EPP1332_0001_0016.A_0022_EPP1332_0001_0017.A_0023_EPP1342_0001_0016.A_0024_EPP1342_0001_0017.A_0026_EPP1518_0002_0017.DIG_Inputs_Device.Status/Error_channel_1 <-> DIG Inputs Device/Status/Error channel 1
//     PlcTask Inputs/GVL_iXlinker.EtherCAT_Master_EPPxxxx.Beckhoff_EPP1xxx.Beckhoff_EPP1xxxEK1122.A_0018_EPP1321_0060_0016.A_0019_EPP1322_0001_0016.A_0020_EPP1322_0001_0017.A_0021_EPP1332_0001_0016.A_0022_EPP1332_0001_0017.A_0023_EPP1342_0001_0016.A_0024_EPP1342_0001_0017.A_0026_EPP1518_0002_0017.DIG_Inputs_Device.Status/Error_channel_2 <-> DIG Inputs Device/Status/Error channel 2
//     PlcTask Inputs/GVL_iXlinker.EtherCAT_Master_EPPxxxx.Beckhoff_EPP1xxx.Beckhoff_EPP1xxxEK1122.A_0018_EPP1321_0060_0016.A_0019_EPP1322_0001_0016.A_0020_EPP1322_0001_0017.A_0021_EPP1332_0001_0016.A_0022_EPP1332_0001_0017.A_0023_EPP1342_0001_0016.A_0024_EPP1342_0001_0017.A_0026_EPP1518_0002_0017.DIG_Inputs_Device.Status/Sync_error <-> DIG Inputs Device/Status/Sync error
//     PlcTask Inputs/GVL_iXlinker.EtherCAT_Master_EPPxxxx.Beckhoff_EPP1xxx.Beckhoff_EPP1xxxEK1122.A_0018_EPP1321_0060_0016.A_0019_EPP1322_0001_0016.A_0020_EPP1322_0001_0017.A_0021_EPP1332_0001_0016.A_0022_EPP1332_0001_0017.A_0023_EPP1342_0001_0016.A_0024_EPP1342_0001_0017.A_0026_EPP1518_0002_0017.DIG_Inputs_Device.Status/TxPDO_State <-> DIG Inputs Device/Status/TxPDO State
//     PlcTask Inputs/GVL_iXlinker.EtherCAT_Master_EPPxxxx.Beckhoff_EPP1xxx.Beckhoff_EPP1xxxEK1122.A_0018_EPP1321_0060_0016.A_0019_EPP1322_0001_0016.A_0020_EPP1322_0001_0017.A_0021_EPP1332_0001_0016.A_0022_EPP1332_0001_0017.A_0023_EPP1342_0001_0016.A_0024_EPP1342_0001_0017.A_0026_EPP1518_0002_0017.DIG_Inputs_Device.Status/TxPDO_Toggle <-> DIG Inputs Device/Status/TxPDO Toggle
//     PlcTask Outputs/GVL_iXlinker.EtherCAT_Master_EPPxxxx.Beckhoff_EPP1xxx.Beckhoff_EPP1xxxEK1122.A_0018_EPP1321_0060_0016.A_0019_EPP1322_0001_0016.A_0020_EPP1322_0001_0017.A_0021_EPP1332_0001_0016.A_0022_EPP1332_0001_0017.A_0023_EPP1342_0001_0016.A_0024_EPP1342_0001_0017.A_0026_EPP1518_0002_0017.CNT_Output_Channel_1.Control/Set_counter <-> CNT Output Channel 1/Control/Set counter
//     PlcTask Outputs/GVL_iXlinker.EtherCAT_Master_EPPxxxx.Beckhoff_EPP1xxx.Beckhoff_EPP1xxxEK1122.A_0018_EPP1321_0060_0016.A_0019_EPP1322_0001_0016.A_0020_EPP1322_0001_0017.A_0021_EPP1332_0001_0016.A_0022_EPP1332_0001_0017.A_0023_EPP1342_0001_0016.A_0024_EPP1342_0001_0017.A_0026_EPP1518_0002_0017.CNT_Output_Channel_2.Control/Set_counter <-> CNT Output Channel 2/Control/Set counter
//     PlcTask Outputs/GVL_iXlinker.EtherCAT_Master_EPPxxxx.Beckhoff_EPP1xxx.Beckhoff_EPP1xxxEK1122.A_0018_EPP1321_0060_0016.A_0019_EPP1322_0001_0016.A_0020_EPP1322_0001_0017.A_0021_EPP1332_0001_0016.A_0022_EPP1332_0001_0017.A_0023_EPP1342_0001_0016.A_0024_EPP1342_0001_0017.A_0026_EPP1518_0002_0017.CNT_Output_Channel_1.Control/Inhibit_counter <-> CNT Output Channel 1/Control/Inhibit counter
//     PlcTask Outputs/GVL_iXlinker.EtherCAT_Master_EPPxxxx.Beckhoff_EPP1xxx.Beckhoff_EPP1xxxEK1122.A_0018_EPP1321_0060_0016.A_0019_EPP1322_0001_0016.A_0020_EPP1322_0001_0017.A_0021_EPP1332_0001_0016.A_0022_EPP1332_0001_0017.A_0023_EPP1342_0001_0016.A_0024_EPP1342_0001_0017.A_0026_EPP1518_0002_0017.CNT_Output_Channel_2.Control/Inhibit_counter <-> CNT Output Channel 2/Control/Inhibit counter
//     PlcTask Outputs/GVL_iXlinker.EtherCAT_Master_EPPxxxx.Beckhoff_EPP1xxx.Beckhoff_EPP1xxxEK1122.A_0018_EPP1321_0060_0016.A_0019_EPP1322_0001_0016.A_0020_EPP1322_0001_0017.A_0021_EPP1332_0001_0016.A_0022_EPP1332_0001_0017.A_0023_EPP1342_0001_0016.A_0024_EPP1342_0001_0017.A_0026_EPP1518_0002_0017.CNT_Output_Channel_1.Set_counter_value <-> CNT Output Channel 1/Set counter value
//     PlcTask Outputs/GVL_iXlinker.EtherCAT_Master_EPPxxxx.Beckhoff_EPP1xxx.Beckhoff_EPP1xxxEK1122.A_0018_EPP1321_0060_0016.A_0019_EPP1322_0001_0016.A_0020_EPP1322_0001_0017.A_0021_EPP1332_0001_0016.A_0022_EPP1332_0001_0017.A_0023_EPP1342_0001_0016.A_0024_EPP1342_0001_0017.A_0026_EPP1518_0002_0017.CNT_Output_Channel_2.Set_counter_value <-> CNT Output Channel 2/Set counter value
//     PlcTask Inputs/GVL_iXlinker.EtherCAT_Master_EPPxxxx.Beckhoff_EPP1xxx.Beckhoff_EPP1xxxEK1122.A_0018_EPP1321_0060_0016.A_0019_EPP1322_0001_0016.A_0020_EPP1322_0001_0017.A_0021_EPP1332_0001_0016.A_0022_EPP1332_0001_0017.A_0023_EPP1342_0001_0016.A_0024_EPP1342_0001_0017.A_0026_EPP1518_0002_0017.WcState.WcState <-> WcState/WcState
//     PlcTask Inputs/GVL_iXlinker.EtherCAT_Master_EPPxxxx.Beckhoff_EPP1xxx.Beckhoff_EPP1xxxEK1122.A_0018_EPP1321_0060_0016.A_0019_EPP1322_0001_0016.A_0020_EPP1322_0001_0017.A_0021_EPP1332_0001_0016.A_0022_EPP1332_0001_0017.A_0023_EPP1342_0001_0016.A_0024_EPP1342_0001_0017.A_0026_EPP1518_0002_0017.WcState.InputToggle <-> WcState/InputToggle
//     PlcTask Inputs/GVL_iXlinker.EtherCAT_Master_EPPxxxx.Beckhoff_EPP1xxx.Beckhoff_EPP1xxxEK1122.A_0018_EPP1321_0060_0016.A_0019_EPP1322_0001_0016.A_0020_EPP1322_0001_0017.A_0021_EPP1332_0001_0016.A_0022_EPP1332_0001_0017.A_0023_EPP1342_0001_0016.A_0024_EPP1342_0001_0017.A_0026_EPP1518_0002_0017.InfoData.AdsAddr <-> InfoData/AdsAddr
//     PlcTask Inputs/GVL_iXlinker.EtherCAT_Master_EPPxxxx.Beckhoff_EPP1xxx.Beckhoff_EPP1xxxEK1122.A_0018_EPP1321_0060_0016.A_0019_EPP1322_0001_0016.A_0020_EPP1322_0001_0017.A_0021_EPP1332_0001_0016.A_0022_EPP1332_0001_0017.A_0023_EPP1342_0001_0016.A_0024_EPP1342_0001_0017.A_0026_EPP1518_0002_0017.InfoData.State <-> InfoData/State
//   PLC/PLC Instance <-> EtherCAT Master EPPxxxx/Beckhoff EPP1xxx/Beckhoff EPP1xxxEK1122/A_0018(EPP1321-0060-0016)/A_0019(EPP1322-0001-0016)/A_0020(EPP1322-0001-0017)/A_0021(EPP1332-0001-0016)/A_0022(EPP1332-0001-0017)/A_0023(EPP1342-0001-0016)/A_0024(EPP1342-0001-0017)/A_0027(EPP1809-0021-0016)
//     PlcTask Inputs/GVL_iXlinker.EtherCAT_Master_EPPxxxx.Beckhoff_EPP1xxx.Beckhoff_EPP1xxxEK1122.A_0018_EPP1321_0060_0016.A_0019_EPP1322_0001_0016.A_0020_EPP1322_0001_0017.A_0021_EPP1332_0001_0016.A_0022_EPP1332_0001_0017.A_0023_EPP1342_0001_0016.A_0024_EPP1342_0001_0017.A_0027_EPP1809_0021_0016.Channel_1.Input <-> Channel 1/Input
//     PlcTask Inputs/GVL_iXlinker.EtherCAT_Master_EPPxxxx.Beckhoff_EPP1xxx.Beckhoff_EPP1xxxEK1122.A_0018_EPP1321_0060_0016.A_0019_EPP1322_0001_0016.A_0020_EPP1322_0001_0017.A_0021_EPP1332_0001_0016.A_0022_EPP1332_0001_0017.A_0023_EPP1342_0001_0016.A_0024_EPP1342_0001_0017.A_0027_EPP1809_0021_0016.Channel_2.Input <-> Channel 2/Input
//     PlcTask Inputs/GVL_iXlinker.EtherCAT_Master_EPPxxxx.Beckhoff_EPP1xxx.Beckhoff_EPP1xxxEK1122.A_0018_EPP1321_0060_0016.A_0019_EPP1322_0001_0016.A_0020_EPP1322_0001_0017.A_0021_EPP1332_0001_0016.A_0022_EPP1332_0001_0017.A_0023_EPP1342_0001_0016.A_0024_EPP1342_0001_0017.A_0027_EPP1809_0021_0016.Channel_3.Input <-> Channel 3/Input
//     PlcTask Inputs/GVL_iXlinker.EtherCAT_Master_EPPxxxx.Beckhoff_EPP1xxx.Beckhoff_EPP1xxxEK1122.A_0018_EPP1321_0060_0016.A_0019_EPP1322_0001_0016.A_0020_EPP1322_0001_0017.A_0021_EPP1332_0001_0016.A_0022_EPP1332_0001_0017.A_0023_EPP1342_0001_0016.A_0024_EPP1342_0001_0017.A_0027_EPP1809_0021_0016.Channel_4.Input <-> Channel 4/Input
//     PlcTask Inputs/GVL_iXlinker.EtherCAT_Master_EPPxxxx.Beckhoff_EPP1xxx.Beckhoff_EPP1xxxEK1122.A_0018_EPP1321_0060_0016.A_0019_EPP1322_0001_0016.A_0020_EPP1322_0001_0017.A_0021_EPP1332_0001_0016.A_0022_EPP1332_0001_0017.A_0023_EPP1342_0001_0016.A_0024_EPP1342_0001_0017.A_0027_EPP1809_0021_0016.Channel_5.Input <-> Channel 5/Input
//     PlcTask Inputs/GVL_iXlinker.EtherCAT_Master_EPPxxxx.Beckhoff_EPP1xxx.Beckhoff_EPP1xxxEK1122.A_0018_EPP1321_0060_0016.A_0019_EPP1322_0001_0016.A_0020_EPP1322_0001_0017.A_0021_EPP1332_0001_0016.A_0022_EPP1332_0001_0017.A_0023_EPP1342_0001_0016.A_0024_EPP1342_0001_0017.A_0027_EPP1809_0021_0016.Channel_6.Input <-> Channel 6/Input
//     PlcTask Inputs/GVL_iXlinker.EtherCAT_Master_EPPxxxx.Beckhoff_EPP1xxx.Beckhoff_EPP1xxxEK1122.A_0018_EPP1321_0060_0016.A_0019_EPP1322_0001_0016.A_0020_EPP1322_0001_0017.A_0021_EPP1332_0001_0016.A_0022_EPP1332_0001_0017.A_0023_EPP1342_0001_0016.A_0024_EPP1342_0001_0017.A_0027_EPP1809_0021_0016.Channel_7.Input <-> Channel 7/Input
//     PlcTask Inputs/GVL_iXlinker.EtherCAT_Master_EPPxxxx.Beckhoff_EPP1xxx.Beckhoff_EPP1xxxEK1122.A_0018_EPP1321_0060_0016.A_0019_EPP1322_0001_0016.A_0020_EPP1322_0001_0017.A_0021_EPP1332_0001_0016.A_0022_EPP1332_0001_0017.A_0023_EPP1342_0001_0016.A_0024_EPP1342_0001_0017.A_0027_EPP1809_0021_0016.Channel_8.Input <-> Channel 8/Input
//     PlcTask Inputs/GVL_iXlinker.EtherCAT_Master_EPPxxxx.Beckhoff_EPP1xxx.Beckhoff_EPP1xxxEK1122.A_0018_EPP1321_0060_0016.A_0019_EPP1322_0001_0016.A_0020_EPP1322_0001_0017.A_0021_EPP1332_0001_0016.A_0022_EPP1332_0001_0017.A_0023_EPP1342_0001_0016.A_0024_EPP1342_0001_0017.A_0027_EPP1809_0021_0016.Channel_9.Input <-> Channel 9/Input
//     PlcTask Inputs/GVL_iXlinker.EtherCAT_Master_EPPxxxx.Beckhoff_EPP1xxx.Beckhoff_EPP1xxxEK1122.A_0018_EPP1321_0060_0016.A_0019_EPP1322_0001_0016.A_0020_EPP1322_0001_0017.A_0021_EPP1332_0001_0016.A_0022_EPP1332_0001_0017.A_0023_EPP1342_0001_0016.A_0024_EPP1342_0001_0017.A_0027_EPP1809_0021_0016.Channel_10.Input <-> Channel 10/Input
//     PlcTask Inputs/GVL_iXlinker.EtherCAT_Master_EPPxxxx.Beckhoff_EPP1xxx.Beckhoff_EPP1xxxEK1122.A_0018_EPP1321_0060_0016.A_0019_EPP1322_0001_0016.A_0020_EPP1322_0001_0017.A_0021_EPP1332_0001_0016.A_0022_EPP1332_0001_0017.A_0023_EPP1342_0001_0016.A_0024_EPP1342_0001_0017.A_0027_EPP1809_0021_0016.Channel_11.Input <-> Channel 11/Input
//     PlcTask Inputs/GVL_iXlinker.EtherCAT_Master_EPPxxxx.Beckhoff_EPP1xxx.Beckhoff_EPP1xxxEK1122.A_0018_EPP1321_0060_0016.A_0019_EPP1322_0001_0016.A_0020_EPP1322_0001_0017.A_0021_EPP1332_0001_0016.A_0022_EPP1332_0001_0017.A_0023_EPP1342_0001_0016.A_0024_EPP1342_0001_0017.A_0027_EPP1809_0021_0016.Channel_12.Input <-> Channel 12/Input
//     PlcTask Inputs/GVL_iXlinker.EtherCAT_Master_EPPxxxx.Beckhoff_EPP1xxx.Beckhoff_EPP1xxxEK1122.A_0018_EPP1321_0060_0016.A_0019_EPP1322_0001_0016.A_0020_EPP1322_0001_0017.A_0021_EPP1332_0001_0016.A_0022_EPP1332_0001_0017.A_0023_EPP1342_0001_0016.A_0024_EPP1342_0001_0017.A_0027_EPP1809_0021_0016.Channel_13.Input <-> Channel 13/Input
//     PlcTask Inputs/GVL_iXlinker.EtherCAT_Master_EPPxxxx.Beckhoff_EPP1xxx.Beckhoff_EPP1xxxEK1122.A_0018_EPP1321_0060_0016.A_0019_EPP1322_0001_0016.A_0020_EPP1322_0001_0017.A_0021_EPP1332_0001_0016.A_0022_EPP1332_0001_0017.A_0023_EPP1342_0001_0016.A_0024_EPP1342_0001_0017.A_0027_EPP1809_0021_0016.Channel_14.Input <-> Channel 14/Input
//     PlcTask Inputs/GVL_iXlinker.EtherCAT_Master_EPPxxxx.Beckhoff_EPP1xxx.Beckhoff_EPP1xxxEK1122.A_0018_EPP1321_0060_0016.A_0019_EPP1322_0001_0016.A_0020_EPP1322_0001_0017.A_0021_EPP1332_0001_0016.A_0022_EPP1332_0001_0017.A_0023_EPP1342_0001_0016.A_0024_EPP1342_0001_0017.A_0027_EPP1809_0021_0016.Channel_15.Input <-> Channel 15/Input
//     PlcTask Inputs/GVL_iXlinker.EtherCAT_Master_EPPxxxx.Beckhoff_EPP1xxx.Beckhoff_EPP1xxxEK1122.A_0018_EPP1321_0060_0016.A_0019_EPP1322_0001_0016.A_0020_EPP1322_0001_0017.A_0021_EPP1332_0001_0016.A_0022_EPP1332_0001_0017.A_0023_EPP1342_0001_0016.A_0024_EPP1342_0001_0017.A_0027_EPP1809_0021_0016.Channel_16.Input <-> Channel 16/Input
